// TIA Portal V16 program export: 3 tag tables, 0 data types, 6 data blocks, 22 code blocks (in call order from the OBs), 35 instance data blocks

VAR_GLOBAL   // PLC tag table "Default tag table"
   EDGE_1 AT %M100.0 : Bool;
   EDGE_2 AT %M100.1 : Bool;
   System_Byte AT %MB1 : Byte;
   FirstScan AT %M1.0 : Bool;
   DiagStatusUpdate AT %M1.1 : Bool;
   AlwaysTRUE AT %M1.2 : Bool;
   AlwaysFALSE AT %M1.3 : Bool;
   Clock_Byte AT %MB0 : Byte;
   Clock_10Hz AT %M0.0 : Bool;
   Clock_5Hz AT %M0.1 : Bool;
   "Clock_2.5Hz" AT %M0.2 : Bool;
   Clock_2Hz AT %M0.3 : Bool;
   "Clock_1.25Hz" AT %M0.4 : Bool;
   Clock_1Hz AT %M0.5 : Bool;
   "Clock_0.625Hz" AT %M0.6 : Bool;
   "Clock_0.5Hz" AT %M0.7 : Bool;
   EDGE_3 AT %M100.2 : Bool;
   EDGE_4 AT %M100.3 : Bool;
   RET_VAL_SYSTEM_TIME AT %MW102 : Word;
   EDGE_5 AT %M100.4 : Bool;
   EDGE_6 AT %M100.5 : Bool;
   EDGE_7 AT %M100.6 : Bool;
END_VAR

VAR_GLOBAL   // PLC tag table "Inputs"
   "EV1.1_ABERTA" AT %I0.0 : Bool;
   "EV1.1_FECHADA" AT %I0.1 : Bool;
   "EV2.1_ABERTA" AT %I0.2 : Bool;
   "EV2.1_FECHADA" AT %I0.3 : Bool;
   "EV3.1_ABERTA" AT %I0.4 : Bool;
   "EV3.1_FECHADA" AT %I0.5 : Bool;
   "EV4.1_ABERTA" AT %I0.6 : Bool;
   "EV4.1_FECHADA" AT %I0.7 : Bool;
   "EV5.1_ABERTA" AT %I1.0 : Bool;
   "EV5.1_FECHADA" AT %I1.1 : Bool;
   "EV1.2_ABERTA" AT %I1.2 : Bool;
   "EV1.2_FECHADA" AT %I1.3 : Bool;
   "EV2.2_ABERTA" AT %I1.4 : Bool;
   "EV2.2_FECHADA" AT %I1.5 : Bool;
   "EV3.2_ABERTA" AT %I2.0 : Bool;
   "EV3.2_FECHADA" AT %I2.1 : Bool;
   "EV4.2_ABERTA" AT %I2.2 : Bool;
   "EV4.2_FECHADA" AT %I2.3 : Bool;
   "EV5.2_ABERTA" AT %I2.4 : Bool;
   "EV5.2_FECHADA" AT %I2.5 : Bool;
   PRESSOSTATO_1 AT %IW4 : Word;
   PRESSOSTATO_2 AT %IW6 : Word;
   AVARIA_BOMBA_1 AT %I2.6 : Bool;
   AVARIA_BOMBA_2 AT %I2.7 : Bool;
   AVARIA_BOMBA_3 AT %I3.0 : Bool;
END_VAR

VAR_GLOBAL   // PLC tag table "Outputs"
   "EV1.1" AT %Q0.0 : Bool;
   "EV2.1" AT %Q0.1 : Bool;
   "EV3.1" AT %Q0.2 : Bool;
   "EV4.1" AT %Q0.3 : Bool;
   "EV5.1" AT %Q0.4 : Bool;
   "EV1.2" AT %Q0.5 : Bool;
   "EV2.2" AT %Q0.6 : Bool;
   "EV3.2" AT %Q0.7 : Bool;
   "EV4.2" AT %Q1.0 : Bool;
   "EV5.2" AT %Q1.1 : Bool;
   BOMBA_1_VAR AT %Q2.0 : Bool;
   BOMBA_2_VAR AT %Q2.1 : Bool;
   BOMBA_3_RESERVA AT %Q2.2 : Bool;
   ULTRAVIOLETA AT %Q2.3 : Bool;
END_VAR

DATA_BLOCK "Dados_Bombas"   // DB11
{ S7_Optimized_Access := 'TRUE' }
VERSION : 0.1
// stored: AutoNumber true, IsOnlyStoredInLoadMemory false, IsRetainMemResEnabled false, IsWriteProtectedInAS false, MemoryReserve 100
   VAR
      CONV_T_ALTERNANCIA_BOMBAS : Time;
      HORAS_TON_B2 : Int;
      HORAS_TON_B3 : Int;
      HORAS_TON_B1 : Int;
   END_VAR
BEGIN
END_DATA_BLOCK

DATA_BLOCK "Estados_HMI"   // DB18
{ S7_Optimized_Access := 'TRUE' }
VERSION : 0.1
// stored: AutoNumber true, IsOnlyStoredInLoadMemory false, IsRetainMemResEnabled false, IsWriteProtectedInAS false, MemoryReserve 100
   VAR
      "EV1.1_ESTADO" : Int;
      "EV2.1_ESTADO" : Int;
      "EV3.1_ESTADO" : Int;
      "EV4.1_ESTADO" : Int;
      "EV5.1_ESTADO" : Int;
      "EV1.2_ESTADO" : Int;
      "EV2.2_ESTADO" : Int;
      "EV3.2_ESTADO" : Int;
      "EV4.2_ESTADO" : Int;
      "EV5.2_ESTADO" : Int;
      "EV1.1_ESTADO_PAGCMD" : Int;
      "EV2.1_ESTADO_PAGCMD" : Int;
      "EV3.1_ESTADO_PAGCMD" : Int;
      "EV4.1_ESTADO_PAGCMD" : Int;
      "EV5.1_ESTADO_PAGCMD" : Int;
      "EV1.2_ESTADO_PAGCMD" : Int;
      "EV2.2_ESTADO_PAGCMD" : Int;
      "EV3.2_ESTADO_PAGCMD" : Int;
      "EV4.2_ESTADO_PAGCMD" : Int;
      "EV5.2_ESTADO_PAGCMD" : Int;
      BOMBA_1_ESTADO : Int;
      BOMBA_2_ESTADO : Int;
      BOMBA_3_ESTADO : Int;
      BOMBA_1_ESTADO_PAGCMD : Int;
      BOMBA_2_ESTADO_PAGCMD : Int;
      BOMBA_3_ESTADO_PAGCMD : Int;
      T_LAV_MINUTOS : Int;
      T_RINSE_MINUTOS : Int;
      ALARMES_LISTA_1 : Word;
      ALARMES_LISTA_2 : Word;
      ALARMES_LISTA_3 : Word;
   END_VAR
BEGIN
END_DATA_BLOCK

DATA_BLOCK "Inputs_HMI"   // DB6
{ S7_Optimized_Access := 'TRUE' }
VERSION : 0.1
// stored: AutoNumber true, IsOnlyStoredInLoadMemory false, IsRetainMemResEnabled false, IsWriteProtectedInAS false, MemoryReserve 100
   VAR RETAIN
      T_LAVAGEM : Time;
      T_RINSE : Time;
      T_STOP_BOMBAS : Time;
      T_POS_EVS : Time;
      ENABLE_CICLO_FILT1 : Bool;
      ENABLE_CICLO_FILT2 : Bool;
   END_VAR
   VAR
      START_CICLO_FILT1 : Bool;
      START_CICLO_FILT2 : Bool;
      STOP_CICLO : Bool;
      REARME : Bool;
      "MAN/AUTO" : Bool;
      "ON_OFF_EV1.1" : Bool;
      "ON_OFF_EV2.1" : Bool;
      "ON_OFF_EV3.1" : Bool;
      "ON_OFF_EV4.1" : Bool;
      "ON_OFF_EV5.1" : Bool;
      "ON_OFF_EV1.2" : Bool;
      "ON_OFF_EV2.2" : Bool;
      "ON_OFF_EV3.2" : Bool;
      "ON_OFF_EV4.2" : Bool;
      "ON_OFF_EV5.2" : Bool;
   END_VAR
   VAR RETAIN
      "MAN/AUTO_BOMBAS" : Bool;
      T_ALTERNANCIA_BOMBAS : Real;
   END_VAR
   VAR
      ON_OFF_BOMBA_1 : Bool;
      ON_OFF_BOMBA_2 : Bool;
      ON_OFF_BOMBA_3 : Bool;
      RESET_CNT_B1 : Bool;
      RESET_CNT_B2 : Bool;
      RESET_CNT_B3 : Bool;
   END_VAR
   VAR RETAIN
      SP_PRESS_FILT1 : Real;
      SP_PRESS_FILT2 : Real;
   END_VAR
BEGIN
END_DATA_BLOCK

DATA_BLOCK "Dados_Ciclo"   // DB7
{ S7_Optimized_Access := 'TRUE' }
VERSION : 0.1
// stored: AutoNumber true, IsOnlyStoredInLoadMemory false, IsRetainMemResEnabled false, IsWriteProtectedInAS false, MemoryReserve 100
   VAR
      HOLD_ETAPA_1 : Bool;
   END_VAR
   VAR RETAIN
      FILTRO1_EM_CICLO : Bool;
      FILTRO2_EM_CICLO : Bool;
      FECHO_FILT_1 : Bool;
      FECHO_FILT_2 : Bool;
      ETAPA_ANTERIOR : Int := 1;
   END_VAR
   VAR
      ETAPA_N : Bool;
      POS_EVS_FILT_1 : String;
      POS_EVS_FILT_2 : String;
      PRESS_SP_FILT_1 : Bool;
      PRESS_SP_FILT_2 : Bool;
   END_VAR
   VAR RETAIN
      STOP_CICLO : Bool;
   END_VAR
   VAR
      AGEND_FILT_1 : Bool;
      AGEND_FILT_2 : Bool;
   END_VAR
   VAR RETAIN
      HORA_INIC_FILT_1 : USInt;
      MIN_INIC_FILT_1 : USInt;
      HORA_INIC_FILT_2 : USInt;
      MIN_INIC_FILT_2 : USInt;
      ENABLE_AGEND_FILT_1 : Bool;
      ENABLE_AGEND_FILT_2 : Bool;
   END_VAR
   VAR
      PRESSÃO_FILT1 : Real;
      PRESSÃO_FILT2 : Real;
   END_VAR
BEGIN
END_DATA_BLOCK

DATA_BLOCK "Etapas_Grafcet"   // DB1
{ S7_Optimized_Access := 'TRUE' }
VERSION : 0.1
// stored: AutoNumber true, IsOnlyStoredInLoadMemory false, IsRetainMemResEnabled false, IsWriteProtectedInAS false, MemoryReserve 100
   VAR
      ETAPA_1 : Bool;
      ETAPA_2 : Bool;
      ETAPA_3 : Bool;
      ETAPA_4 : Bool;
      ETAPA_5 : Bool;
      ETAPA_6 : Bool;
      ETAPA_7 : Bool;
      ETAPA_8 : Bool;
      ETAPA_9 : Bool;
      ETAPA_10 : Bool;
      ETAPA_11 : Bool;
      ETAPA_12 : Bool;
      ETAPA_13 : Bool;
      ETAPA_14 : Bool;
      ETAPA_15 : Bool := true;
      ETAPA_16 : Bool;
   END_VAR
BEGIN
END_DATA_BLOCK

DATA_BLOCK "System_Time"   // DB40
{ S7_Optimized_Access := 'TRUE' }
VERSION : 0.1
// stored: AutoNumber true, IsOnlyStoredInLoadMemory false, IsRetainMemResEnabled false, IsWriteProtectedInAS false, MemoryReserve 100
   VAR
      REAL_TIME_DATA : DTL;
   END_VAR
BEGIN
END_DATA_BLOCK

ORGANIZATION_BLOCK "Main"   // OB1, LAD, ProgramCycle
TITLE = "Main Program Sweep (Cycle)"
{ S7_Optimized_Access := 'TRUE' }
VERSION : 0.1
// stored: AutoNumber true, IsIECCheckEnabled false, SetENOAutomatically false
   VAR_INPUT
      Initial_Call : Bool;   // Initial call of this OB
      Remanence : Bool;   // =True, if remanent data are available
   END_VAR
   VAR_TEMP   // added for the SCL form of the ladder/FBD networks
      _w1 : Bool;
   END_VAR
BEGIN

REGION Network 1: Ciclo de lavagem e enxaguamento
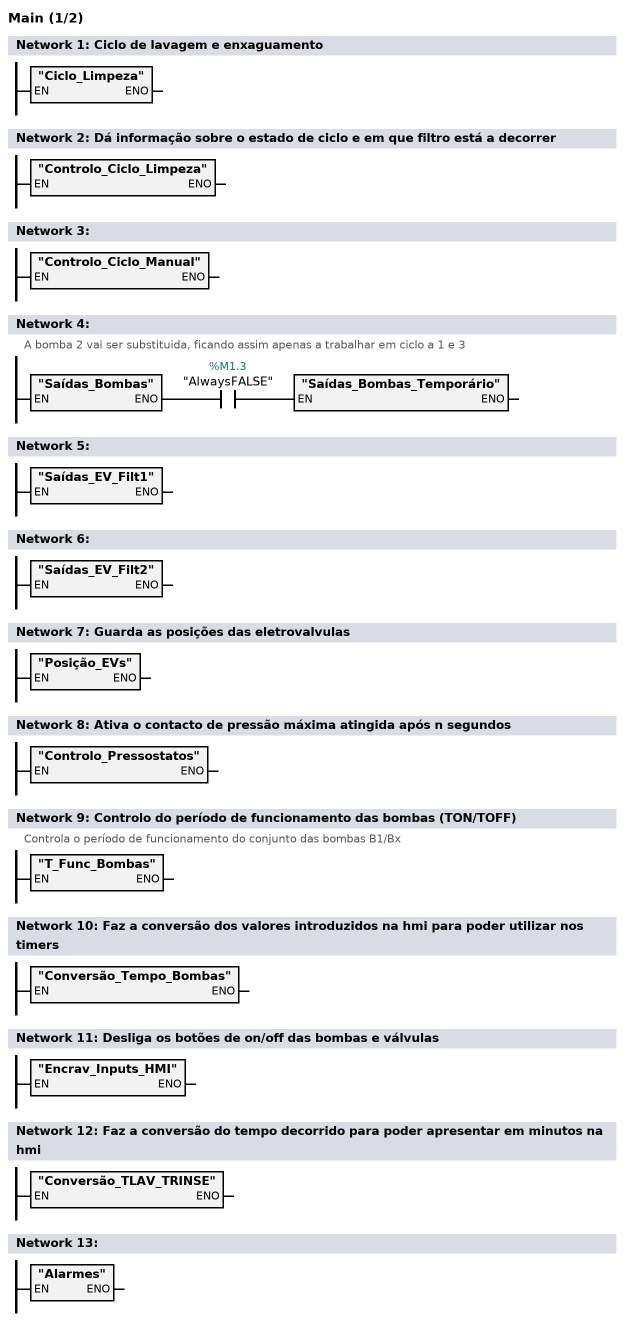
   RUNG wire#powerrail
      "Ciclo_Limpeza"()
   END_RUNG
   // the same network as SCL:
   "Ciclo_Limpeza"();
END_REGION

REGION Network 2: Dá informação sobre o estado de ciclo e em que filtro está a decorrer
   RUNG wire#powerrail
      "Controlo_Ciclo_Limpeza"()
   END_RUNG
   // the same network as SCL:
   "Controlo_Ciclo_Limpeza"();
END_REGION

REGION Network 3
   RUNG wire#powerrail
      "Controlo_Ciclo_Manual"()
   END_RUNG
   // the same network as SCL:
   "Controlo_Ciclo_Manual"();
END_REGION

REGION Network 4
   // A bomba 2 vai ser substituida, ficando assim apenas a trabalhar em ciclo a 1 e 3
   RUNG wire#powerrail
      "Saídas_Bombas"()
      Contact( "AlwaysFALSE" )
      "Saídas_Bombas_Temporário"()
   END_RUNG
   // the same network as SCL:
   "Saídas_Bombas"(ENO => #_w1);
   IF #_w1 AND "AlwaysFALSE" THEN "Saídas_Bombas_Temporário"(); END_IF;
END_REGION

REGION Network 5
   RUNG wire#powerrail
      "Saídas_EV_Filt1"()
   END_RUNG
   // the same network as SCL:
   "Saídas_EV_Filt1"();
END_REGION

REGION Network 6
   RUNG wire#powerrail
      "Saídas_EV_Filt2"()
   END_RUNG
   // the same network as SCL:
   "Saídas_EV_Filt2"();
END_REGION

REGION Network 7: Guarda as posições das eletrovalvulas
   RUNG wire#powerrail
      "Posição_EVs"()
   END_RUNG
   // the same network as SCL:
   "Posição_EVs"();
END_REGION

REGION Network 8: Ativa o contacto de pressão máxima atingida após n segundos
   RUNG wire#powerrail
      "Controlo_Pressostatos"()
   END_RUNG
   // the same network as SCL:
   "Controlo_Pressostatos"();
END_REGION

REGION Network 9: Controlo do período de funcionamento das bombas (TON/TOFF)
   // Controla o período de funcionamento do conjunto das bombas B1/Bx
   RUNG wire#powerrail
      "T_Func_Bombas"()
   END_RUNG
   // the same network as SCL:
   "T_Func_Bombas"();
END_REGION

REGION Network 10: Faz a conversão dos valores introduzidos na hmi para poder utilizar nos timers
   RUNG wire#powerrail
      "Conversão_Tempo_Bombas"()
   END_RUNG
   // the same network as SCL:
   "Conversão_Tempo_Bombas"();
END_REGION

REGION Network 11: Desliga os botões de on/off das bombas e válvulas
   RUNG wire#powerrail
      "Encrav_Inputs_HMI"()
   END_RUNG
   // the same network as SCL:
   "Encrav_Inputs_HMI"();
END_REGION

REGION Network 12: Faz a conversão do tempo decorrido para poder apresentar em minutos na hmi
   RUNG wire#powerrail
      "Conversão_TLAV_TRINSE"()
   END_RUNG
   // the same network as SCL:
   "Conversão_TLAV_TRINSE"();
END_REGION

REGION Network 13
   RUNG wire#powerrail
      "Alarmes"()
   END_RUNG
   // the same network as SCL:
   "Alarmes"();
END_REGION

REGION Network 14: Ultravioleta
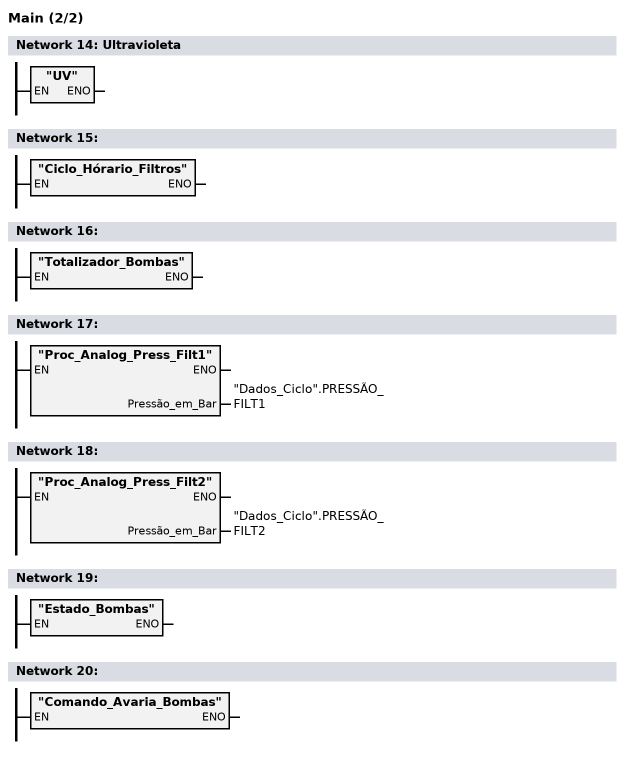
   RUNG wire#powerrail
      "UV"()
   END_RUNG
   // the same network as SCL:
   "UV"();
END_REGION

REGION Network 15
   RUNG wire#powerrail
      "Ciclo_Hórario_Filtros"()
   END_RUNG
   // the same network as SCL:
   "Ciclo_Hórario_Filtros"();
END_REGION

REGION Network 16
   RUNG wire#powerrail
      "Totalizador_Bombas"()
   END_RUNG
   // the same network as SCL:
   "Totalizador_Bombas"();
END_REGION

REGION Network 17
   RUNG wire#powerrail
      "Proc_Analog_Press_Filt1"(Pressão_em_Bar => "Dados_Ciclo".PRESSÃO_FILT1)
   END_RUNG
   // the same network as SCL:
   "Proc_Analog_Press_Filt1"(Pressão_em_Bar => "Dados_Ciclo".PRESSÃO_FILT1);
END_REGION

REGION Network 18
   RUNG wire#powerrail
      "Proc_Analog_Press_Filt2"(Pressão_em_Bar => "Dados_Ciclo".PRESSÃO_FILT2)
   END_RUNG
   // the same network as SCL:
   "Proc_Analog_Press_Filt2"(Pressão_em_Bar => "Dados_Ciclo".PRESSÃO_FILT2);
END_REGION

REGION Network 19
   RUNG wire#powerrail
      "Estado_Bombas"()
   END_RUNG
   // the same network as SCL:
   "Estado_Bombas"();
END_REGION

REGION Network 20
   RUNG wire#powerrail
      "Comando_Avaria_Bombas"()
   END_RUNG
   // the same network as SCL:
   "Comando_Avaria_Bombas"();
END_REGION
END_ORGANIZATION_BLOCK

FUNCTION "Ciclo_Limpeza" : Void   // FC1, LAD
TITLE = Ciclo de lavagem e enxaguamento
{ S7_Optimized_Access := 'TRUE' }
VERSION : 0.1
// stored: AutoNumber true, IsIECCheckEnabled false, SetENOAutomatically false, UDAEnableTagReadback false
   VAR_TEMP   // added for the SCL form of the ladder/FBD networks
      _w1 : Bool;
      _w2 : Bool;
      _w3 : Bool;
   END_VAR
BEGIN

REGION Network 1: Etapa 1 (Início)
   // Início com EV's na posição de filtração. As bombas podem estar ligadas ou não, conforme a posição do switch 4
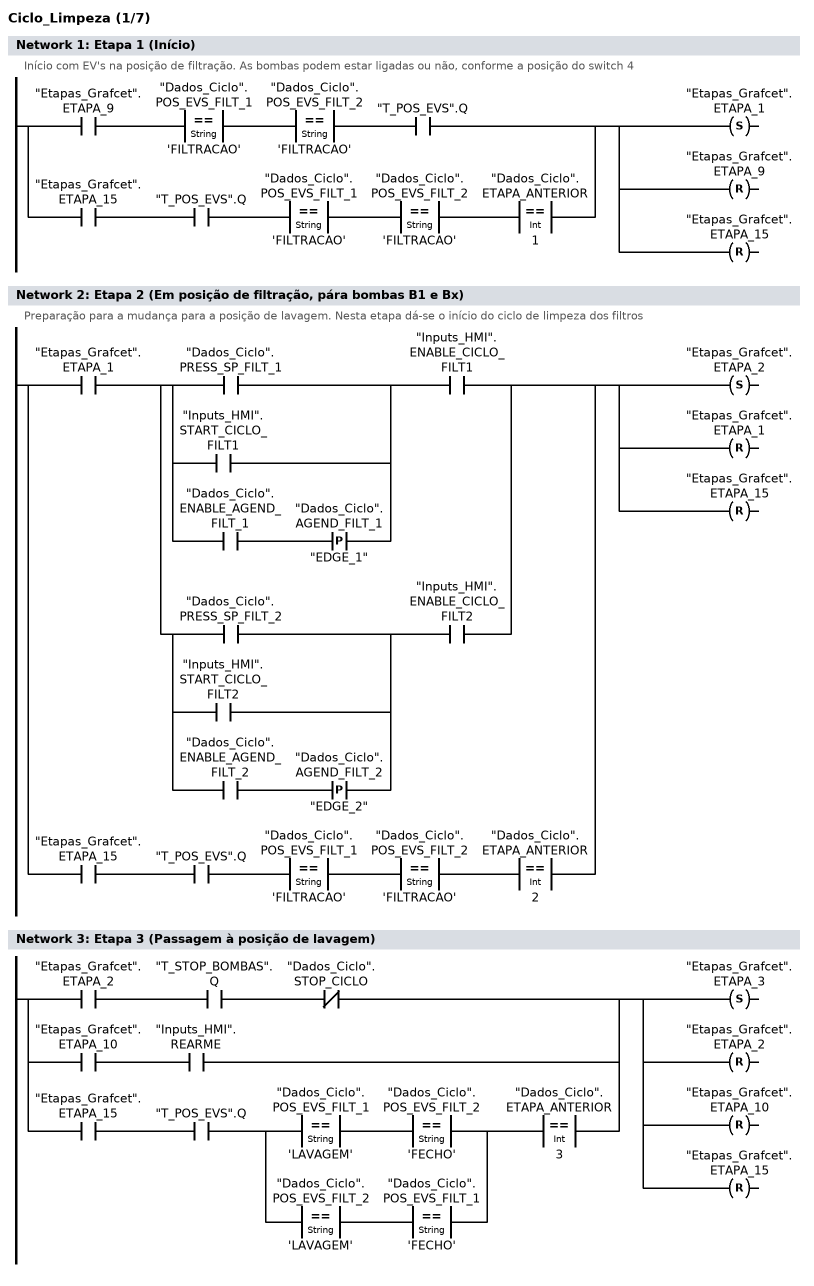
   RUNG wire#powerrail
      Contact( "Etapas_Grafcet".ETAPA_9 )
      { S7_Templates := "SrcType := String" } EQ_Contact(in1 := "Dados_Ciclo".POS_EVS_FILT_1, in2 := 'FILTRACAO')
      { S7_Templates := "SrcType := String" } EQ_Contact(in1 := "Dados_Ciclo".POS_EVS_FILT_2, in2 := 'FILTRACAO')
      Contact( "T_POS_EVS".Q )
      wire#w1
      S_Coil( "Etapas_Grafcet".ETAPA_1 )
   END_RUNG
   RUNG wire#powerrail
      Contact( "Etapas_Grafcet".ETAPA_15 )
      Contact( "T_POS_EVS".Q )
      { S7_Templates := "SrcType := String" } EQ_Contact(in1 := "Dados_Ciclo".POS_EVS_FILT_1, in2 := 'FILTRACAO')
      { S7_Templates := "SrcType := String" } EQ_Contact(in1 := "Dados_Ciclo".POS_EVS_FILT_2, in2 := 'FILTRACAO')
      { S7_Templates := "SrcType := Int" } EQ_Contact(in1 := "Dados_Ciclo".ETAPA_ANTERIOR, in2 := 1)
   END_RUNG wire#w1
   RUNG wire#w1
      R_Coil( "Etapas_Grafcet".ETAPA_9 )
   END_RUNG
   RUNG wire#w1
      R_Coil( "Etapas_Grafcet".ETAPA_15 )
   END_RUNG
   // the same network as SCL:
   IF ("Etapas_Grafcet".ETAPA_9 AND ("Dados_Ciclo".POS_EVS_FILT_1 = 'FILTRACAO') AND ("Dados_Ciclo".POS_EVS_FILT_2 = 'FILTRACAO') AND "T_POS_EVS".Q) OR ("Etapas_Grafcet".ETAPA_15 AND "T_POS_EVS".Q AND ("Dados_Ciclo".POS_EVS_FILT_1 = 'FILTRACAO') AND ("Dados_Ciclo".POS_EVS_FILT_2 = 'FILTRACAO') AND ("Dados_Ciclo".ETAPA_ANTERIOR = 1)) THEN
       "Etapas_Grafcet".ETAPA_1 := TRUE;
   END_IF;
   #_w1 := ("Etapas_Grafcet".ETAPA_9 AND ("Dados_Ciclo".POS_EVS_FILT_1 = 'FILTRACAO') AND ("Dados_Ciclo".POS_EVS_FILT_2 = 'FILTRACAO') AND "T_POS_EVS".Q) OR ("Etapas_Grafcet".ETAPA_15 AND "T_POS_EVS".Q AND ("Dados_Ciclo".POS_EVS_FILT_1 = 'FILTRACAO') AND ("Dados_Ciclo".POS_EVS_FILT_2 = 'FILTRACAO') AND ("Dados_Ciclo".ETAPA_ANTERIOR = 1));
   IF #_w1 THEN
       "Etapas_Grafcet".ETAPA_9 := FALSE;
       "Etapas_Grafcet".ETAPA_15 := FALSE;
   END_IF;
END_REGION

REGION Network 2: Etapa 2 (Em posição de filtração, pára bombas B1 e Bx)
   // Preparação para a mudança para a posição de lavagem. Nesta etapa dá-se o início do ciclo de limpeza dos filtros
   RUNG wire#powerrail
      Contact( "Etapas_Grafcet".ETAPA_1 )
      wire#w1
      Contact( "Dados_Ciclo".PRESS_SP_FILT_1 )
      wire#w2
      Contact( "Inputs_HMI".ENABLE_CICLO_FILT1 )
      wire#w3
      S_Coil( "Etapas_Grafcet".ETAPA_2 )
   END_RUNG
   RUNG wire#w1
      Contact( "Inputs_HMI".START_CICLO_FILT1 )
   END_RUNG wire#w2
   RUNG wire#w1
      Contact( "Dados_Ciclo".ENABLE_AGEND_FILT_1 )
      P_Contact(operand := "Dados_Ciclo".AGEND_FILT_1, bit := "EDGE_1")
   END_RUNG wire#w2
   RUNG wire#w1
      Contact( "Dados_Ciclo".PRESS_SP_FILT_2 )
      wire#w4
      Contact( "Inputs_HMI".ENABLE_CICLO_FILT2 )
   END_RUNG wire#w3
   RUNG wire#w1
      Contact( "Inputs_HMI".START_CICLO_FILT2 )
   END_RUNG wire#w4
   RUNG wire#w1
      Contact( "Dados_Ciclo".ENABLE_AGEND_FILT_2 )
      P_Contact(operand := "Dados_Ciclo".AGEND_FILT_2, bit := "EDGE_2")
   END_RUNG wire#w4
   RUNG wire#powerrail
      Contact( "Etapas_Grafcet".ETAPA_15 )
      Contact( "T_POS_EVS".Q )
      { S7_Templates := "SrcType := String" } EQ_Contact(in1 := "Dados_Ciclo".POS_EVS_FILT_1, in2 := 'FILTRACAO')
      { S7_Templates := "SrcType := String" } EQ_Contact(in1 := "Dados_Ciclo".POS_EVS_FILT_2, in2 := 'FILTRACAO')
      { S7_Templates := "SrcType := Int" } EQ_Contact(in1 := "Dados_Ciclo".ETAPA_ANTERIOR, in2 := 2)
   END_RUNG wire#w3
   RUNG wire#w3
      R_Coil( "Etapas_Grafcet".ETAPA_1 )
   END_RUNG
   RUNG wire#w3
      R_Coil( "Etapas_Grafcet".ETAPA_15 )
   END_RUNG
   // the same network as SCL:
   #_w1 := "Etapas_Grafcet".ETAPA_1 AND "Dados_Ciclo".ENABLE_AGEND_FILT_1 AND "Dados_Ciclo".AGEND_FILT_1 AND NOT "EDGE_1";   // rising edge of "Dados_Ciclo".AGEND_FILT_1
   "EDGE_1" := "Dados_Ciclo".AGEND_FILT_1;
   #_w2 := "Etapas_Grafcet".ETAPA_1 AND "Dados_Ciclo".ENABLE_AGEND_FILT_2 AND "Dados_Ciclo".AGEND_FILT_2 AND NOT "EDGE_2";   // rising edge of "Dados_Ciclo".AGEND_FILT_2
   "EDGE_2" := "Dados_Ciclo".AGEND_FILT_2;
   IF ((("Etapas_Grafcet".ETAPA_1 AND ("Dados_Ciclo".PRESS_SP_FILT_1 OR "Inputs_HMI".START_CICLO_FILT1)) OR #_w1) AND "Inputs_HMI".ENABLE_CICLO_FILT1) OR ((("Etapas_Grafcet".ETAPA_1 AND ("Dados_Ciclo".PRESS_SP_FILT_2 OR "Inputs_HMI".START_CICLO_FILT2)) OR #_w2) AND "Inputs_HMI".ENABLE_CICLO_FILT2) OR ("Etapas_Grafcet".ETAPA_15 AND "T_POS_EVS".Q AND ("Dados_Ciclo".POS_EVS_FILT_1 = 'FILTRACAO') AND ("Dados_Ciclo".POS_EVS_FILT_2 = 'FILTRACAO') AND ("Dados_Ciclo".ETAPA_ANTERIOR = 2)) THEN
       "Etapas_Grafcet".ETAPA_2 := TRUE;
   END_IF;
   #_w3 := ((("Etapas_Grafcet".ETAPA_1 AND ("Dados_Ciclo".PRESS_SP_FILT_1 OR "Inputs_HMI".START_CICLO_FILT1)) OR #_w1) AND "Inputs_HMI".ENABLE_CICLO_FILT1) OR ((("Etapas_Grafcet".ETAPA_1 AND ("Dados_Ciclo".PRESS_SP_FILT_2 OR "Inputs_HMI".START_CICLO_FILT2)) OR #_w2) AND "Inputs_HMI".ENABLE_CICLO_FILT2) OR ("Etapas_Grafcet".ETAPA_15 AND "T_POS_EVS".Q AND ("Dados_Ciclo".POS_EVS_FILT_1 = 'FILTRACAO') AND ("Dados_Ciclo".POS_EVS_FILT_2 = 'FILTRACAO') AND ("Dados_Ciclo".ETAPA_ANTERIOR = 2));
   IF #_w3 THEN
       "Etapas_Grafcet".ETAPA_1 := FALSE;
       "Etapas_Grafcet".ETAPA_15 := FALSE;
   END_IF;
END_REGION

REGION Network 3: Etapa 3 (Passagem à posição de lavagem)
   RUNG wire#powerrail
      Contact( "Etapas_Grafcet".ETAPA_2 )
      Contact( "T_STOP_BOMBAS".Q )
      I_Contact( "Dados_Ciclo".STOP_CICLO )
      wire#w1
      S_Coil( "Etapas_Grafcet".ETAPA_3 )
   END_RUNG
   RUNG wire#powerrail
      Contact( "Etapas_Grafcet".ETAPA_10 )
      Contact( "Inputs_HMI".REARME )
   END_RUNG wire#w1
   RUNG wire#powerrail
      Contact( "Etapas_Grafcet".ETAPA_15 )
      Contact( "T_POS_EVS".Q )
      wire#w2
      { S7_Templates := "SrcType := String" } EQ_Contact(in1 := "Dados_Ciclo".POS_EVS_FILT_1, in2 := 'LAVAGEM')
      { S7_Templates := "SrcType := String" } EQ_Contact(in1 := "Dados_Ciclo".POS_EVS_FILT_2, in2 := 'FECHO')
      wire#w3
      { S7_Templates := "SrcType := Int" } EQ_Contact(in1 := "Dados_Ciclo".ETAPA_ANTERIOR, in2 := 3)
   END_RUNG wire#w1
   RUNG wire#w2
      { S7_Templates := "SrcType := String" } EQ_Contact(in1 := "Dados_Ciclo".POS_EVS_FILT_2, in2 := 'LAVAGEM')
      { S7_Templates := "SrcType := String" } EQ_Contact(in1 := "Dados_Ciclo".POS_EVS_FILT_1, in2 := 'FECHO')
   END_RUNG wire#w3
   RUNG wire#w1
      R_Coil( "Etapas_Grafcet".ETAPA_2 )
   END_RUNG
   RUNG wire#w1
      R_Coil( "Etapas_Grafcet".ETAPA_10 )
   END_RUNG
   RUNG wire#w1
      R_Coil( "Etapas_Grafcet".ETAPA_15 )
   END_RUNG
   // the same network as SCL:
   IF ("Etapas_Grafcet".ETAPA_2 AND "T_STOP_BOMBAS".Q AND NOT "Dados_Ciclo".STOP_CICLO) OR ("Etapas_Grafcet".ETAPA_10 AND "Inputs_HMI".REARME) OR ("Etapas_Grafcet".ETAPA_15 AND "T_POS_EVS".Q AND ((("Dados_Ciclo".POS_EVS_FILT_1 = 'LAVAGEM') AND ("Dados_Ciclo".POS_EVS_FILT_2 = 'FECHO')) OR (("Dados_Ciclo".POS_EVS_FILT_2 = 'LAVAGEM') AND ("Dados_Ciclo".POS_EVS_FILT_1 = 'FECHO'))) AND ("Dados_Ciclo".ETAPA_ANTERIOR = 3)) THEN
       "Etapas_Grafcet".ETAPA_3 := TRUE;
   END_IF;
   #_w1 := ("Etapas_Grafcet".ETAPA_2 AND "T_STOP_BOMBAS".Q AND NOT "Dados_Ciclo".STOP_CICLO) OR ("Etapas_Grafcet".ETAPA_10 AND "Inputs_HMI".REARME) OR ("Etapas_Grafcet".ETAPA_15 AND "T_POS_EVS".Q AND ((("Dados_Ciclo".POS_EVS_FILT_1 = 'LAVAGEM') AND ("Dados_Ciclo".POS_EVS_FILT_2 = 'FECHO')) OR (("Dados_Ciclo".POS_EVS_FILT_2 = 'LAVAGEM') AND ("Dados_Ciclo".POS_EVS_FILT_1 = 'FECHO'))) AND ("Dados_Ciclo".ETAPA_ANTERIOR = 3));
   IF #_w1 THEN
       "Etapas_Grafcet".ETAPA_2 := FALSE;
       "Etapas_Grafcet".ETAPA_10 := FALSE;
       "Etapas_Grafcet".ETAPA_15 := FALSE;
   END_IF;
END_REGION

REGION Network 4: Etapa 4 (Em lavagem, B1 e BX ligadas)
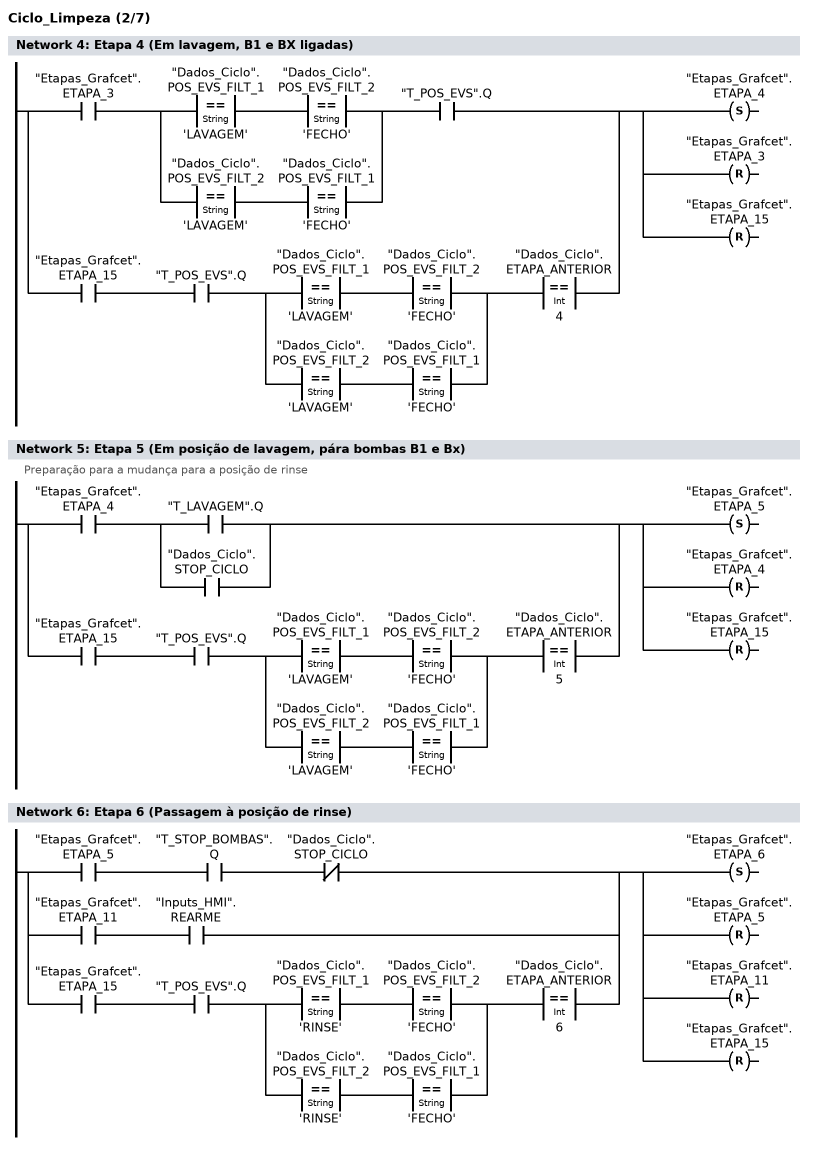
   RUNG wire#powerrail
      Contact( "Etapas_Grafcet".ETAPA_3 )
      wire#w1
      { S7_Templates := "SrcType := String" } EQ_Contact(in1 := "Dados_Ciclo".POS_EVS_FILT_1, in2 := 'LAVAGEM')
      { S7_Templates := "SrcType := String" } EQ_Contact(in1 := "Dados_Ciclo".POS_EVS_FILT_2, in2 := 'FECHO')
      wire#w2
      Contact( "T_POS_EVS".Q )
      wire#w3
      S_Coil( "Etapas_Grafcet".ETAPA_4 )
   END_RUNG
   RUNG wire#w1
      { S7_Templates := "SrcType := String" } EQ_Contact(in1 := "Dados_Ciclo".POS_EVS_FILT_2, in2 := 'LAVAGEM')
      { S7_Templates := "SrcType := String" } EQ_Contact(in1 := "Dados_Ciclo".POS_EVS_FILT_1, in2 := 'FECHO')
   END_RUNG wire#w2
   RUNG wire#powerrail
      Contact( "Etapas_Grafcet".ETAPA_15 )
      Contact( "T_POS_EVS".Q )
      wire#w4
      { S7_Templates := "SrcType := String" } EQ_Contact(in1 := "Dados_Ciclo".POS_EVS_FILT_1, in2 := 'LAVAGEM')
      { S7_Templates := "SrcType := String" } EQ_Contact(in1 := "Dados_Ciclo".POS_EVS_FILT_2, in2 := 'FECHO')
      wire#w5
      { S7_Templates := "SrcType := Int" } EQ_Contact(in1 := "Dados_Ciclo".ETAPA_ANTERIOR, in2 := 4)
   END_RUNG wire#w3
   RUNG wire#w4
      { S7_Templates := "SrcType := String" } EQ_Contact(in1 := "Dados_Ciclo".POS_EVS_FILT_2, in2 := 'LAVAGEM')
      { S7_Templates := "SrcType := String" } EQ_Contact(in1 := "Dados_Ciclo".POS_EVS_FILT_1, in2 := 'FECHO')
   END_RUNG wire#w5
   RUNG wire#w3
      R_Coil( "Etapas_Grafcet".ETAPA_3 )
   END_RUNG
   RUNG wire#w3
      R_Coil( "Etapas_Grafcet".ETAPA_15 )
   END_RUNG
   // the same network as SCL:
   IF ("Etapas_Grafcet".ETAPA_3 AND ((("Dados_Ciclo".POS_EVS_FILT_1 = 'LAVAGEM') AND ("Dados_Ciclo".POS_EVS_FILT_2 = 'FECHO')) OR (("Dados_Ciclo".POS_EVS_FILT_2 = 'LAVAGEM') AND ("Dados_Ciclo".POS_EVS_FILT_1 = 'FECHO'))) AND "T_POS_EVS".Q) OR ("Etapas_Grafcet".ETAPA_15 AND "T_POS_EVS".Q AND ((("Dados_Ciclo".POS_EVS_FILT_1 = 'LAVAGEM') AND ("Dados_Ciclo".POS_EVS_FILT_2 = 'FECHO')) OR (("Dados_Ciclo".POS_EVS_FILT_2 = 'LAVAGEM') AND ("Dados_Ciclo".POS_EVS_FILT_1 = 'FECHO'))) AND ("Dados_Ciclo".ETAPA_ANTERIOR = 4)) THEN
       "Etapas_Grafcet".ETAPA_4 := TRUE;
   END_IF;
   #_w1 := ("Etapas_Grafcet".ETAPA_3 AND ((("Dados_Ciclo".POS_EVS_FILT_1 = 'LAVAGEM') AND ("Dados_Ciclo".POS_EVS_FILT_2 = 'FECHO')) OR (("Dados_Ciclo".POS_EVS_FILT_2 = 'LAVAGEM') AND ("Dados_Ciclo".POS_EVS_FILT_1 = 'FECHO'))) AND "T_POS_EVS".Q) OR ("Etapas_Grafcet".ETAPA_15 AND "T_POS_EVS".Q AND ((("Dados_Ciclo".POS_EVS_FILT_1 = 'LAVAGEM') AND ("Dados_Ciclo".POS_EVS_FILT_2 = 'FECHO')) OR (("Dados_Ciclo".POS_EVS_FILT_2 = 'LAVAGEM') AND ("Dados_Ciclo".POS_EVS_FILT_1 = 'FECHO'))) AND ("Dados_Ciclo".ETAPA_ANTERIOR = 4));
   IF #_w1 THEN
       "Etapas_Grafcet".ETAPA_3 := FALSE;
       "Etapas_Grafcet".ETAPA_15 := FALSE;
   END_IF;
END_REGION

REGION Network 5: Etapa 5 (Em posição de lavagem, pára bombas B1 e Bx)
   // Preparação para a mudança para a posição de rinse
   RUNG wire#powerrail
      Contact( "Etapas_Grafcet".ETAPA_4 )
      wire#w1
      Contact( "T_LAVAGEM".Q )
      wire#w2
      S_Coil( "Etapas_Grafcet".ETAPA_5 )
   END_RUNG
   RUNG wire#w1
      Contact( "Dados_Ciclo".STOP_CICLO )
   END_RUNG wire#w2
   RUNG wire#powerrail
      Contact( "Etapas_Grafcet".ETAPA_15 )
      Contact( "T_POS_EVS".Q )
      wire#w3
      { S7_Templates := "SrcType := String" } EQ_Contact(in1 := "Dados_Ciclo".POS_EVS_FILT_1, in2 := 'LAVAGEM')
      { S7_Templates := "SrcType := String" } EQ_Contact(in1 := "Dados_Ciclo".POS_EVS_FILT_2, in2 := 'FECHO')
      wire#w4
      { S7_Templates := "SrcType := Int" } EQ_Contact(in1 := "Dados_Ciclo".ETAPA_ANTERIOR, in2 := 5)
   END_RUNG wire#w2
   RUNG wire#w3
      { S7_Templates := "SrcType := String" } EQ_Contact(in1 := "Dados_Ciclo".POS_EVS_FILT_2, in2 := 'LAVAGEM')
      { S7_Templates := "SrcType := String" } EQ_Contact(in1 := "Dados_Ciclo".POS_EVS_FILT_1, in2 := 'FECHO')
   END_RUNG wire#w4
   RUNG wire#w2
      R_Coil( "Etapas_Grafcet".ETAPA_4 )
   END_RUNG
   RUNG wire#w2
      R_Coil( "Etapas_Grafcet".ETAPA_15 )
   END_RUNG
   // the same network as SCL:
   IF ("Etapas_Grafcet".ETAPA_4 AND ("T_LAVAGEM".Q OR "Dados_Ciclo".STOP_CICLO)) OR ("Etapas_Grafcet".ETAPA_15 AND "T_POS_EVS".Q AND ((("Dados_Ciclo".POS_EVS_FILT_1 = 'LAVAGEM') AND ("Dados_Ciclo".POS_EVS_FILT_2 = 'FECHO')) OR (("Dados_Ciclo".POS_EVS_FILT_2 = 'LAVAGEM') AND ("Dados_Ciclo".POS_EVS_FILT_1 = 'FECHO'))) AND ("Dados_Ciclo".ETAPA_ANTERIOR = 5)) THEN
       "Etapas_Grafcet".ETAPA_5 := TRUE;
   END_IF;
   #_w1 := ("Etapas_Grafcet".ETAPA_4 AND ("T_LAVAGEM".Q OR "Dados_Ciclo".STOP_CICLO)) OR ("Etapas_Grafcet".ETAPA_15 AND "T_POS_EVS".Q AND ((("Dados_Ciclo".POS_EVS_FILT_1 = 'LAVAGEM') AND ("Dados_Ciclo".POS_EVS_FILT_2 = 'FECHO')) OR (("Dados_Ciclo".POS_EVS_FILT_2 = 'LAVAGEM') AND ("Dados_Ciclo".POS_EVS_FILT_1 = 'FECHO'))) AND ("Dados_Ciclo".ETAPA_ANTERIOR = 5));
   IF #_w1 THEN
       "Etapas_Grafcet".ETAPA_4 := FALSE;
       "Etapas_Grafcet".ETAPA_15 := FALSE;
   END_IF;
END_REGION

REGION Network 6: Etapa 6 (Passagem à posição de rinse)
   RUNG wire#powerrail
      Contact( "Etapas_Grafcet".ETAPA_5 )
      Contact( "T_STOP_BOMBAS".Q )
      I_Contact( "Dados_Ciclo".STOP_CICLO )
      wire#w1
      S_Coil( "Etapas_Grafcet".ETAPA_6 )
   END_RUNG
   RUNG wire#powerrail
      Contact( "Etapas_Grafcet".ETAPA_11 )
      Contact( "Inputs_HMI".REARME )
   END_RUNG wire#w1
   RUNG wire#powerrail
      Contact( "Etapas_Grafcet".ETAPA_15 )
      Contact( "T_POS_EVS".Q )
      wire#w2
      { S7_Templates := "SrcType := String" } EQ_Contact(in1 := "Dados_Ciclo".POS_EVS_FILT_1, in2 := 'RINSE')
      { S7_Templates := "SrcType := String" } EQ_Contact(in1 := "Dados_Ciclo".POS_EVS_FILT_2, in2 := 'FECHO')
      wire#w3
      { S7_Templates := "SrcType := Int" } EQ_Contact(in1 := "Dados_Ciclo".ETAPA_ANTERIOR, in2 := 6)
   END_RUNG wire#w1
   RUNG wire#w2
      { S7_Templates := "SrcType := String" } EQ_Contact(in1 := "Dados_Ciclo".POS_EVS_FILT_2, in2 := 'RINSE')
      { S7_Templates := "SrcType := String" } EQ_Contact(in1 := "Dados_Ciclo".POS_EVS_FILT_1, in2 := 'FECHO')
   END_RUNG wire#w3
   RUNG wire#w1
      R_Coil( "Etapas_Grafcet".ETAPA_5 )
   END_RUNG
   RUNG wire#w1
      R_Coil( "Etapas_Grafcet".ETAPA_11 )
   END_RUNG
   RUNG wire#w1
      R_Coil( "Etapas_Grafcet".ETAPA_15 )
   END_RUNG
   // the same network as SCL:
   IF ("Etapas_Grafcet".ETAPA_5 AND "T_STOP_BOMBAS".Q AND NOT "Dados_Ciclo".STOP_CICLO) OR ("Etapas_Grafcet".ETAPA_11 AND "Inputs_HMI".REARME) OR ("Etapas_Grafcet".ETAPA_15 AND "T_POS_EVS".Q AND ((("Dados_Ciclo".POS_EVS_FILT_1 = 'RINSE') AND ("Dados_Ciclo".POS_EVS_FILT_2 = 'FECHO')) OR (("Dados_Ciclo".POS_EVS_FILT_2 = 'RINSE') AND ("Dados_Ciclo".POS_EVS_FILT_1 = 'FECHO'))) AND ("Dados_Ciclo".ETAPA_ANTERIOR = 6)) THEN
       "Etapas_Grafcet".ETAPA_6 := TRUE;
   END_IF;
   #_w1 := ("Etapas_Grafcet".ETAPA_5 AND "T_STOP_BOMBAS".Q AND NOT "Dados_Ciclo".STOP_CICLO) OR ("Etapas_Grafcet".ETAPA_11 AND "Inputs_HMI".REARME) OR ("Etapas_Grafcet".ETAPA_15 AND "T_POS_EVS".Q AND ((("Dados_Ciclo".POS_EVS_FILT_1 = 'RINSE') AND ("Dados_Ciclo".POS_EVS_FILT_2 = 'FECHO')) OR (("Dados_Ciclo".POS_EVS_FILT_2 = 'RINSE') AND ("Dados_Ciclo".POS_EVS_FILT_1 = 'FECHO'))) AND ("Dados_Ciclo".ETAPA_ANTERIOR = 6));
   IF #_w1 THEN
       "Etapas_Grafcet".ETAPA_5 := FALSE;
       "Etapas_Grafcet".ETAPA_11 := FALSE;
       "Etapas_Grafcet".ETAPA_15 := FALSE;
   END_IF;
END_REGION

REGION Network 7: Etapa 7 (Em rinse, B1 ligada)
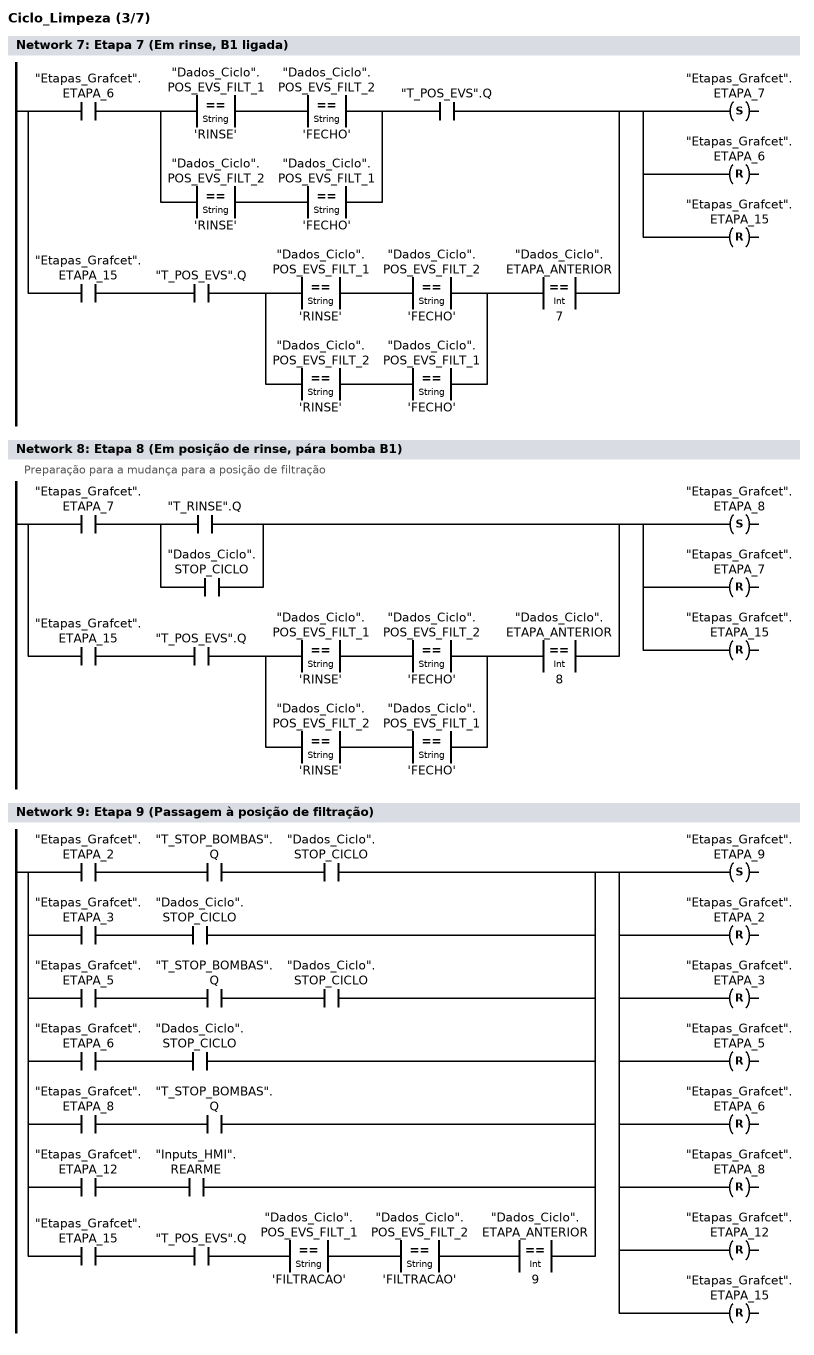
   RUNG wire#powerrail
      Contact( "Etapas_Grafcet".ETAPA_6 )
      wire#w1
      { S7_Templates := "SrcType := String" } EQ_Contact(in1 := "Dados_Ciclo".POS_EVS_FILT_1, in2 := 'RINSE')
      { S7_Templates := "SrcType := String" } EQ_Contact(in1 := "Dados_Ciclo".POS_EVS_FILT_2, in2 := 'FECHO')
      wire#w2
      Contact( "T_POS_EVS".Q )
      wire#w3
      S_Coil( "Etapas_Grafcet".ETAPA_7 )
   END_RUNG
   RUNG wire#w1
      { S7_Templates := "SrcType := String" } EQ_Contact(in1 := "Dados_Ciclo".POS_EVS_FILT_2, in2 := 'RINSE')
      { S7_Templates := "SrcType := String" } EQ_Contact(in1 := "Dados_Ciclo".POS_EVS_FILT_1, in2 := 'FECHO')
   END_RUNG wire#w2
   RUNG wire#powerrail
      Contact( "Etapas_Grafcet".ETAPA_15 )
      Contact( "T_POS_EVS".Q )
      wire#w4
      { S7_Templates := "SrcType := String" } EQ_Contact(in1 := "Dados_Ciclo".POS_EVS_FILT_1, in2 := 'RINSE')
      { S7_Templates := "SrcType := String" } EQ_Contact(in1 := "Dados_Ciclo".POS_EVS_FILT_2, in2 := 'FECHO')
      wire#w5
      { S7_Templates := "SrcType := Int" } EQ_Contact(in1 := "Dados_Ciclo".ETAPA_ANTERIOR, in2 := 7)
   END_RUNG wire#w3
   RUNG wire#w4
      { S7_Templates := "SrcType := String" } EQ_Contact(in1 := "Dados_Ciclo".POS_EVS_FILT_2, in2 := 'RINSE')
      { S7_Templates := "SrcType := String" } EQ_Contact(in1 := "Dados_Ciclo".POS_EVS_FILT_1, in2 := 'FECHO')
   END_RUNG wire#w5
   RUNG wire#w3
      R_Coil( "Etapas_Grafcet".ETAPA_6 )
   END_RUNG
   RUNG wire#w3
      R_Coil( "Etapas_Grafcet".ETAPA_15 )
   END_RUNG
   // the same network as SCL:
   IF ("Etapas_Grafcet".ETAPA_6 AND ((("Dados_Ciclo".POS_EVS_FILT_1 = 'RINSE') AND ("Dados_Ciclo".POS_EVS_FILT_2 = 'FECHO')) OR (("Dados_Ciclo".POS_EVS_FILT_2 = 'RINSE') AND ("Dados_Ciclo".POS_EVS_FILT_1 = 'FECHO'))) AND "T_POS_EVS".Q) OR ("Etapas_Grafcet".ETAPA_15 AND "T_POS_EVS".Q AND ((("Dados_Ciclo".POS_EVS_FILT_1 = 'RINSE') AND ("Dados_Ciclo".POS_EVS_FILT_2 = 'FECHO')) OR (("Dados_Ciclo".POS_EVS_FILT_2 = 'RINSE') AND ("Dados_Ciclo".POS_EVS_FILT_1 = 'FECHO'))) AND ("Dados_Ciclo".ETAPA_ANTERIOR = 7)) THEN
       "Etapas_Grafcet".ETAPA_7 := TRUE;
   END_IF;
   #_w1 := ("Etapas_Grafcet".ETAPA_6 AND ((("Dados_Ciclo".POS_EVS_FILT_1 = 'RINSE') AND ("Dados_Ciclo".POS_EVS_FILT_2 = 'FECHO')) OR (("Dados_Ciclo".POS_EVS_FILT_2 = 'RINSE') AND ("Dados_Ciclo".POS_EVS_FILT_1 = 'FECHO'))) AND "T_POS_EVS".Q) OR ("Etapas_Grafcet".ETAPA_15 AND "T_POS_EVS".Q AND ((("Dados_Ciclo".POS_EVS_FILT_1 = 'RINSE') AND ("Dados_Ciclo".POS_EVS_FILT_2 = 'FECHO')) OR (("Dados_Ciclo".POS_EVS_FILT_2 = 'RINSE') AND ("Dados_Ciclo".POS_EVS_FILT_1 = 'FECHO'))) AND ("Dados_Ciclo".ETAPA_ANTERIOR = 7));
   IF #_w1 THEN
       "Etapas_Grafcet".ETAPA_6 := FALSE;
       "Etapas_Grafcet".ETAPA_15 := FALSE;
   END_IF;
END_REGION

REGION Network 8: Etapa 8 (Em posição de rinse, pára bomba B1)
   // Preparação para a mudança para a posição de filtração
   RUNG wire#powerrail
      Contact( "Etapas_Grafcet".ETAPA_7 )
      wire#w1
      Contact( "T_RINSE".Q )
      wire#w2
      S_Coil( "Etapas_Grafcet".ETAPA_8 )
   END_RUNG
   RUNG wire#w1
      Contact( "Dados_Ciclo".STOP_CICLO )
   END_RUNG wire#w2
   RUNG wire#powerrail
      Contact( "Etapas_Grafcet".ETAPA_15 )
      Contact( "T_POS_EVS".Q )
      wire#w3
      { S7_Templates := "SrcType := String" } EQ_Contact(in1 := "Dados_Ciclo".POS_EVS_FILT_1, in2 := 'RINSE')
      { S7_Templates := "SrcType := String" } EQ_Contact(in1 := "Dados_Ciclo".POS_EVS_FILT_2, in2 := 'FECHO')
      wire#w4
      { S7_Templates := "SrcType := Int" } EQ_Contact(in1 := "Dados_Ciclo".ETAPA_ANTERIOR, in2 := 8)
   END_RUNG wire#w2
   RUNG wire#w3
      { S7_Templates := "SrcType := String" } EQ_Contact(in1 := "Dados_Ciclo".POS_EVS_FILT_2, in2 := 'RINSE')
      { S7_Templates := "SrcType := String" } EQ_Contact(in1 := "Dados_Ciclo".POS_EVS_FILT_1, in2 := 'FECHO')
   END_RUNG wire#w4
   RUNG wire#w2
      R_Coil( "Etapas_Grafcet".ETAPA_7 )
   END_RUNG
   RUNG wire#w2
      R_Coil( "Etapas_Grafcet".ETAPA_15 )
   END_RUNG
   // the same network as SCL:
   IF ("Etapas_Grafcet".ETAPA_7 AND ("T_RINSE".Q OR "Dados_Ciclo".STOP_CICLO)) OR ("Etapas_Grafcet".ETAPA_15 AND "T_POS_EVS".Q AND ((("Dados_Ciclo".POS_EVS_FILT_1 = 'RINSE') AND ("Dados_Ciclo".POS_EVS_FILT_2 = 'FECHO')) OR (("Dados_Ciclo".POS_EVS_FILT_2 = 'RINSE') AND ("Dados_Ciclo".POS_EVS_FILT_1 = 'FECHO'))) AND ("Dados_Ciclo".ETAPA_ANTERIOR = 8)) THEN
       "Etapas_Grafcet".ETAPA_8 := TRUE;
   END_IF;
   #_w1 := ("Etapas_Grafcet".ETAPA_7 AND ("T_RINSE".Q OR "Dados_Ciclo".STOP_CICLO)) OR ("Etapas_Grafcet".ETAPA_15 AND "T_POS_EVS".Q AND ((("Dados_Ciclo".POS_EVS_FILT_1 = 'RINSE') AND ("Dados_Ciclo".POS_EVS_FILT_2 = 'FECHO')) OR (("Dados_Ciclo".POS_EVS_FILT_2 = 'RINSE') AND ("Dados_Ciclo".POS_EVS_FILT_1 = 'FECHO'))) AND ("Dados_Ciclo".ETAPA_ANTERIOR = 8));
   IF #_w1 THEN
       "Etapas_Grafcet".ETAPA_7 := FALSE;
       "Etapas_Grafcet".ETAPA_15 := FALSE;
   END_IF;
END_REGION

REGION Network 9: Etapa 9 (Passagem à posição de filtração)
   RUNG wire#powerrail
      Contact( "Etapas_Grafcet".ETAPA_2 )
      Contact( "T_STOP_BOMBAS".Q )
      Contact( "Dados_Ciclo".STOP_CICLO )
      wire#w1
      S_Coil( "Etapas_Grafcet".ETAPA_9 )
   END_RUNG
   RUNG wire#powerrail
      Contact( "Etapas_Grafcet".ETAPA_3 )
      Contact( "Dados_Ciclo".STOP_CICLO )
   END_RUNG wire#w1
   RUNG wire#powerrail
      Contact( "Etapas_Grafcet".ETAPA_5 )
      Contact( "T_STOP_BOMBAS".Q )
      Contact( "Dados_Ciclo".STOP_CICLO )
   END_RUNG wire#w1
   RUNG wire#powerrail
      Contact( "Etapas_Grafcet".ETAPA_6 )
      Contact( "Dados_Ciclo".STOP_CICLO )
   END_RUNG wire#w1
   RUNG wire#powerrail
      Contact( "Etapas_Grafcet".ETAPA_8 )
      Contact( "T_STOP_BOMBAS".Q )
   END_RUNG wire#w1
   RUNG wire#powerrail
      Contact( "Etapas_Grafcet".ETAPA_12 )
      Contact( "Inputs_HMI".REARME )
   END_RUNG wire#w1
   RUNG wire#powerrail
      Contact( "Etapas_Grafcet".ETAPA_15 )
      Contact( "T_POS_EVS".Q )
      { S7_Templates := "SrcType := String" } EQ_Contact(in1 := "Dados_Ciclo".POS_EVS_FILT_1, in2 := 'FILTRACAO')
      { S7_Templates := "SrcType := String" } EQ_Contact(in1 := "Dados_Ciclo".POS_EVS_FILT_2, in2 := 'FILTRACAO')
      { S7_Templates := "SrcType := Int" } EQ_Contact(in1 := "Dados_Ciclo".ETAPA_ANTERIOR, in2 := 9)
   END_RUNG wire#w1
   RUNG wire#w1
      R_Coil( "Etapas_Grafcet".ETAPA_2 )
   END_RUNG
   RUNG wire#w1
      R_Coil( "Etapas_Grafcet".ETAPA_3 )
   END_RUNG
   RUNG wire#w1
      R_Coil( "Etapas_Grafcet".ETAPA_5 )
   END_RUNG
   RUNG wire#w1
      R_Coil( "Etapas_Grafcet".ETAPA_6 )
   END_RUNG
   RUNG wire#w1
      R_Coil( "Etapas_Grafcet".ETAPA_8 )
   END_RUNG
   RUNG wire#w1
      R_Coil( "Etapas_Grafcet".ETAPA_12 )
   END_RUNG
   RUNG wire#w1
      R_Coil( "Etapas_Grafcet".ETAPA_15 )
   END_RUNG
   // the same network as SCL:
   IF ("Etapas_Grafcet".ETAPA_2 AND "T_STOP_BOMBAS".Q AND "Dados_Ciclo".STOP_CICLO) OR ("Etapas_Grafcet".ETAPA_3 AND "Dados_Ciclo".STOP_CICLO) OR ("Etapas_Grafcet".ETAPA_5 AND "T_STOP_BOMBAS".Q AND "Dados_Ciclo".STOP_CICLO) OR ("Etapas_Grafcet".ETAPA_6 AND "Dados_Ciclo".STOP_CICLO) OR ("Etapas_Grafcet".ETAPA_8 AND "T_STOP_BOMBAS".Q) OR ("Etapas_Grafcet".ETAPA_12 AND "Inputs_HMI".REARME) OR ("Etapas_Grafcet".ETAPA_15 AND "T_POS_EVS".Q AND ("Dados_Ciclo".POS_EVS_FILT_1 = 'FILTRACAO') AND ("Dados_Ciclo".POS_EVS_FILT_2 = 'FILTRACAO') AND ("Dados_Ciclo".ETAPA_ANTERIOR = 9)) THEN
       "Etapas_Grafcet".ETAPA_9 := TRUE;
   END_IF;
   #_w1 := ("Etapas_Grafcet".ETAPA_2 AND "T_STOP_BOMBAS".Q AND "Dados_Ciclo".STOP_CICLO) OR ("Etapas_Grafcet".ETAPA_3 AND "Dados_Ciclo".STOP_CICLO) OR ("Etapas_Grafcet".ETAPA_5 AND "T_STOP_BOMBAS".Q AND "Dados_Ciclo".STOP_CICLO) OR ("Etapas_Grafcet".ETAPA_6 AND "Dados_Ciclo".STOP_CICLO) OR ("Etapas_Grafcet".ETAPA_8 AND "T_STOP_BOMBAS".Q) OR ("Etapas_Grafcet".ETAPA_12 AND "Inputs_HMI".REARME) OR ("Etapas_Grafcet".ETAPA_15 AND "T_POS_EVS".Q AND ("Dados_Ciclo".POS_EVS_FILT_1 = 'FILTRACAO') AND ("Dados_Ciclo".POS_EVS_FILT_2 = 'FILTRACAO') AND ("Dados_Ciclo".ETAPA_ANTERIOR = 9));
   IF #_w1 THEN
       "Etapas_Grafcet".ETAPA_2 := FALSE;
       "Etapas_Grafcet".ETAPA_3 := FALSE;
       "Etapas_Grafcet".ETAPA_5 := FALSE;
       "Etapas_Grafcet".ETAPA_6 := FALSE;
       "Etapas_Grafcet".ETAPA_8 := FALSE;
       "Etapas_Grafcet".ETAPA_12 := FALSE;
       "Etapas_Grafcet".ETAPA_15 := FALSE;
   END_IF;
END_REGION

REGION Network 10: ETAPA 10 (Alarme posição lavagem)
   // As ev's não estão na posição de lavagem / fecho
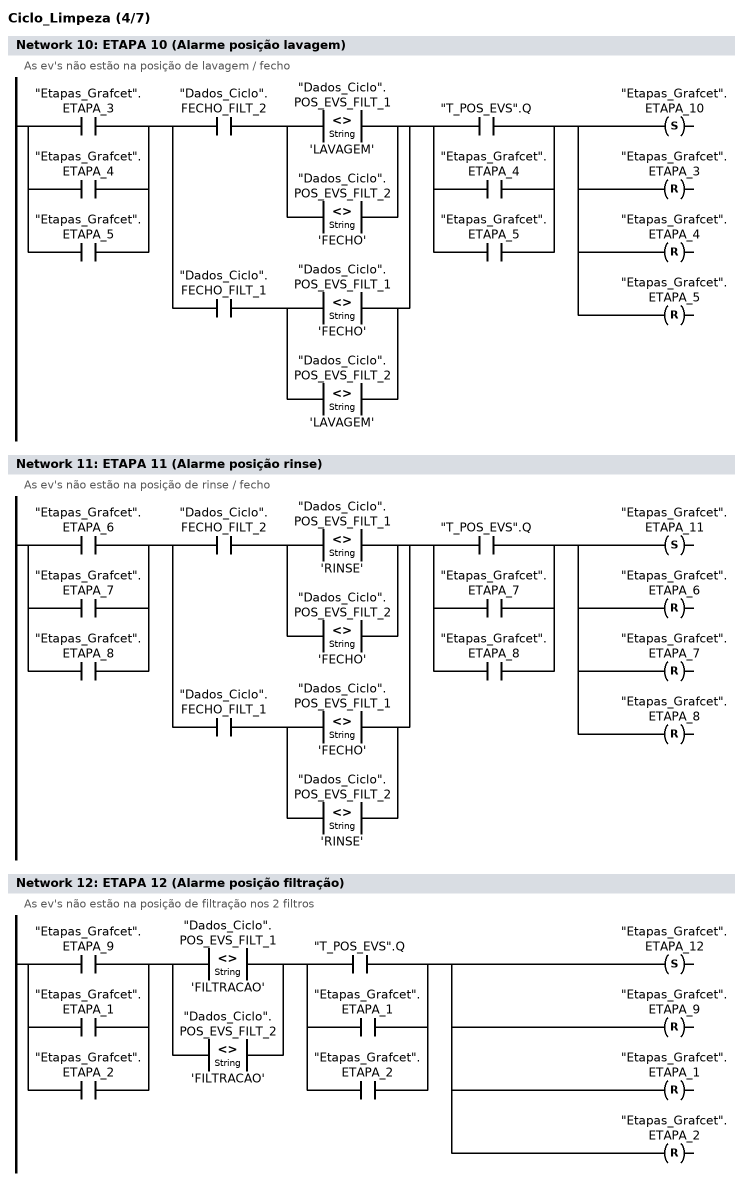
   RUNG wire#powerrail
      Contact( "Etapas_Grafcet".ETAPA_3 )
      wire#w1
      Contact( "Dados_Ciclo".FECHO_FILT_2 )
      wire#w2
      { S7_Templates := "SrcType := String" } NE_Contact(in1 := "Dados_Ciclo".POS_EVS_FILT_1, in2 := 'LAVAGEM')
      wire#w3
      Contact( "T_POS_EVS".Q )
      wire#w5
      S_Coil( "Etapas_Grafcet".ETAPA_10 )
   END_RUNG
   RUNG wire#powerrail
      Contact( "Etapas_Grafcet".ETAPA_4 )
   END_RUNG wire#w1
   RUNG wire#powerrail
      Contact( "Etapas_Grafcet".ETAPA_5 )
   END_RUNG wire#w1
   RUNG wire#w2
      { S7_Templates := "SrcType := String" } NE_Contact(in1 := "Dados_Ciclo".POS_EVS_FILT_2, in2 := 'FECHO')
   END_RUNG wire#w3
   RUNG wire#w1
      Contact( "Dados_Ciclo".FECHO_FILT_1 )
      wire#w4
      { S7_Templates := "SrcType := String" } NE_Contact(in1 := "Dados_Ciclo".POS_EVS_FILT_1, in2 := 'FECHO')
   END_RUNG wire#w3
   RUNG wire#w4
      { S7_Templates := "SrcType := String" } NE_Contact(in1 := "Dados_Ciclo".POS_EVS_FILT_2, in2 := 'LAVAGEM')
   END_RUNG wire#w3
   RUNG wire#w3
      Contact( "Etapas_Grafcet".ETAPA_4 )
   END_RUNG wire#w5
   RUNG wire#w3
      Contact( "Etapas_Grafcet".ETAPA_5 )
   END_RUNG wire#w5
   RUNG wire#w5
      R_Coil( "Etapas_Grafcet".ETAPA_3 )
   END_RUNG
   RUNG wire#w5
      R_Coil( "Etapas_Grafcet".ETAPA_4 )
   END_RUNG
   RUNG wire#w5
      R_Coil( "Etapas_Grafcet".ETAPA_5 )
   END_RUNG
   // the same network as SCL:
   IF ("Etapas_Grafcet".ETAPA_3 OR "Etapas_Grafcet".ETAPA_4 OR "Etapas_Grafcet".ETAPA_5) AND (("Dados_Ciclo".FECHO_FILT_2 AND (("Dados_Ciclo".POS_EVS_FILT_1 <> 'LAVAGEM') OR ("Dados_Ciclo".POS_EVS_FILT_2 <> 'FECHO'))) OR ("Dados_Ciclo".FECHO_FILT_1 AND (("Dados_Ciclo".POS_EVS_FILT_1 <> 'FECHO') OR ("Dados_Ciclo".POS_EVS_FILT_2 <> 'LAVAGEM')))) AND ("T_POS_EVS".Q OR "Etapas_Grafcet".ETAPA_4 OR "Etapas_Grafcet".ETAPA_5) THEN
       "Etapas_Grafcet".ETAPA_10 := TRUE;
   END_IF;
   #_w1 := ("Etapas_Grafcet".ETAPA_3 OR "Etapas_Grafcet".ETAPA_4 OR "Etapas_Grafcet".ETAPA_5) AND (("Dados_Ciclo".FECHO_FILT_2 AND (("Dados_Ciclo".POS_EVS_FILT_1 <> 'LAVAGEM') OR ("Dados_Ciclo".POS_EVS_FILT_2 <> 'FECHO'))) OR ("Dados_Ciclo".FECHO_FILT_1 AND (("Dados_Ciclo".POS_EVS_FILT_1 <> 'FECHO') OR ("Dados_Ciclo".POS_EVS_FILT_2 <> 'LAVAGEM')))) AND ("T_POS_EVS".Q OR "Etapas_Grafcet".ETAPA_4 OR "Etapas_Grafcet".ETAPA_5);
   IF #_w1 THEN
       "Etapas_Grafcet".ETAPA_3 := FALSE;
       "Etapas_Grafcet".ETAPA_4 := FALSE;
       "Etapas_Grafcet".ETAPA_5 := FALSE;
   END_IF;
END_REGION

REGION Network 11: ETAPA 11 (Alarme posição rinse)
   // As ev's não estão na posição de rinse / fecho
   RUNG wire#powerrail
      Contact( "Etapas_Grafcet".ETAPA_6 )
      wire#w1
      Contact( "Dados_Ciclo".FECHO_FILT_2 )
      wire#w2
      { S7_Templates := "SrcType := String" } NE_Contact(in1 := "Dados_Ciclo".POS_EVS_FILT_1, in2 := 'RINSE')
      wire#w3
      Contact( "T_POS_EVS".Q )
      wire#w5
      S_Coil( "Etapas_Grafcet".ETAPA_11 )
   END_RUNG
   RUNG wire#powerrail
      Contact( "Etapas_Grafcet".ETAPA_7 )
   END_RUNG wire#w1
   RUNG wire#powerrail
      Contact( "Etapas_Grafcet".ETAPA_8 )
   END_RUNG wire#w1
   RUNG wire#w2
      { S7_Templates := "SrcType := String" } NE_Contact(in1 := "Dados_Ciclo".POS_EVS_FILT_2, in2 := 'FECHO')
   END_RUNG wire#w3
   RUNG wire#w1
      Contact( "Dados_Ciclo".FECHO_FILT_1 )
      wire#w4
      { S7_Templates := "SrcType := String" } NE_Contact(in1 := "Dados_Ciclo".POS_EVS_FILT_1, in2 := 'FECHO')
   END_RUNG wire#w3
   RUNG wire#w4
      { S7_Templates := "SrcType := String" } NE_Contact(in1 := "Dados_Ciclo".POS_EVS_FILT_2, in2 := 'RINSE')
   END_RUNG wire#w3
   RUNG wire#w3
      Contact( "Etapas_Grafcet".ETAPA_7 )
   END_RUNG wire#w5
   RUNG wire#w3
      Contact( "Etapas_Grafcet".ETAPA_8 )
   END_RUNG wire#w5
   RUNG wire#w5
      R_Coil( "Etapas_Grafcet".ETAPA_6 )
   END_RUNG
   RUNG wire#w5
      R_Coil( "Etapas_Grafcet".ETAPA_7 )
   END_RUNG
   RUNG wire#w5
      R_Coil( "Etapas_Grafcet".ETAPA_8 )
   END_RUNG
   // the same network as SCL:
   IF ("Etapas_Grafcet".ETAPA_6 OR "Etapas_Grafcet".ETAPA_7 OR "Etapas_Grafcet".ETAPA_8) AND (("Dados_Ciclo".FECHO_FILT_2 AND (("Dados_Ciclo".POS_EVS_FILT_1 <> 'RINSE') OR ("Dados_Ciclo".POS_EVS_FILT_2 <> 'FECHO'))) OR ("Dados_Ciclo".FECHO_FILT_1 AND (("Dados_Ciclo".POS_EVS_FILT_1 <> 'FECHO') OR ("Dados_Ciclo".POS_EVS_FILT_2 <> 'RINSE')))) AND ("T_POS_EVS".Q OR "Etapas_Grafcet".ETAPA_7 OR "Etapas_Grafcet".ETAPA_8) THEN
       "Etapas_Grafcet".ETAPA_11 := TRUE;
   END_IF;
   #_w1 := ("Etapas_Grafcet".ETAPA_6 OR "Etapas_Grafcet".ETAPA_7 OR "Etapas_Grafcet".ETAPA_8) AND (("Dados_Ciclo".FECHO_FILT_2 AND (("Dados_Ciclo".POS_EVS_FILT_1 <> 'RINSE') OR ("Dados_Ciclo".POS_EVS_FILT_2 <> 'FECHO'))) OR ("Dados_Ciclo".FECHO_FILT_1 AND (("Dados_Ciclo".POS_EVS_FILT_1 <> 'FECHO') OR ("Dados_Ciclo".POS_EVS_FILT_2 <> 'RINSE')))) AND ("T_POS_EVS".Q OR "Etapas_Grafcet".ETAPA_7 OR "Etapas_Grafcet".ETAPA_8);
   IF #_w1 THEN
       "Etapas_Grafcet".ETAPA_6 := FALSE;
       "Etapas_Grafcet".ETAPA_7 := FALSE;
       "Etapas_Grafcet".ETAPA_8 := FALSE;
   END_IF;
END_REGION

REGION Network 12: ETAPA 12 (Alarme posição filtração)
   // As ev's não estão na posição de filtração nos 2 filtros
   RUNG wire#powerrail
      Contact( "Etapas_Grafcet".ETAPA_9 )
      wire#w1
      { S7_Templates := "SrcType := String" } NE_Contact(in1 := "Dados_Ciclo".POS_EVS_FILT_1, in2 := 'FILTRACAO')
      wire#w2
      Contact( "T_POS_EVS".Q )
      wire#w3
      S_Coil( "Etapas_Grafcet".ETAPA_12 )
   END_RUNG
   RUNG wire#powerrail
      Contact( "Etapas_Grafcet".ETAPA_1 )
   END_RUNG wire#w1
   RUNG wire#powerrail
      Contact( "Etapas_Grafcet".ETAPA_2 )
   END_RUNG wire#w1
   RUNG wire#w1
      { S7_Templates := "SrcType := String" } NE_Contact(in1 := "Dados_Ciclo".POS_EVS_FILT_2, in2 := 'FILTRACAO')
   END_RUNG wire#w2
   RUNG wire#w2
      Contact( "Etapas_Grafcet".ETAPA_1 )
   END_RUNG wire#w3
   RUNG wire#w2
      Contact( "Etapas_Grafcet".ETAPA_2 )
   END_RUNG wire#w3
   RUNG wire#w3
      R_Coil( "Etapas_Grafcet".ETAPA_9 )
   END_RUNG
   RUNG wire#w3
      R_Coil( "Etapas_Grafcet".ETAPA_1 )
   END_RUNG
   RUNG wire#w3
      R_Coil( "Etapas_Grafcet".ETAPA_2 )
   END_RUNG
   // the same network as SCL:
   IF ("Etapas_Grafcet".ETAPA_9 OR "Etapas_Grafcet".ETAPA_1 OR "Etapas_Grafcet".ETAPA_2) AND (("Dados_Ciclo".POS_EVS_FILT_1 <> 'FILTRACAO') OR ("Dados_Ciclo".POS_EVS_FILT_2 <> 'FILTRACAO')) AND ("T_POS_EVS".Q OR "Etapas_Grafcet".ETAPA_1 OR "Etapas_Grafcet".ETAPA_2) THEN
       "Etapas_Grafcet".ETAPA_12 := TRUE;
   END_IF;
   #_w1 := ("Etapas_Grafcet".ETAPA_9 OR "Etapas_Grafcet".ETAPA_1 OR "Etapas_Grafcet".ETAPA_2) AND (("Dados_Ciclo".POS_EVS_FILT_1 <> 'FILTRACAO') OR ("Dados_Ciclo".POS_EVS_FILT_2 <> 'FILTRACAO')) AND ("T_POS_EVS".Q OR "Etapas_Grafcet".ETAPA_1 OR "Etapas_Grafcet".ETAPA_2);
   IF #_w1 THEN
       "Etapas_Grafcet".ETAPA_9 := FALSE;
       "Etapas_Grafcet".ETAPA_1 := FALSE;
       "Etapas_Grafcet".ETAPA_2 := FALSE;
   END_IF;
END_REGION

REGION Network 13: Etapa 13 (Preparação para modo manual)
   // A etapa_n são as etapas de 1 a 9. A etapa 13 corresponde à preparação para entrada em manual. Param as bombas e mantém a posição das válvulas da etapa anterior. O reset às etapas de 1 a 9 é feito em Controlo_Ciclo_Manual
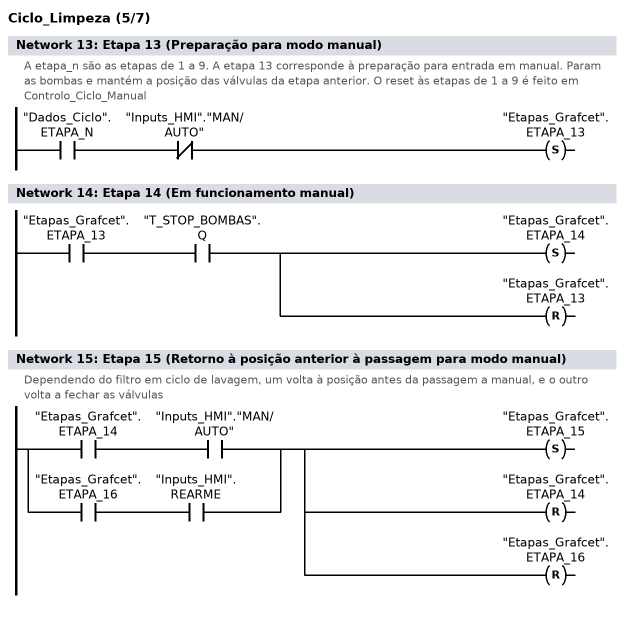
   RUNG wire#powerrail
      Contact( "Dados_Ciclo".ETAPA_N )
      I_Contact( "Inputs_HMI"."MAN/AUTO" )
      S_Coil( "Etapas_Grafcet".ETAPA_13 )
   END_RUNG
   // the same network as SCL:
   IF "Dados_Ciclo".ETAPA_N AND NOT "Inputs_HMI"."MAN/AUTO" THEN "Etapas_Grafcet".ETAPA_13 := TRUE; END_IF;
END_REGION

REGION Network 14: Etapa 14 (Em funcionamento manual)
   RUNG wire#powerrail
      Contact( "Etapas_Grafcet".ETAPA_13 )
      Contact( "T_STOP_BOMBAS".Q )
      wire#w1
      S_Coil( "Etapas_Grafcet".ETAPA_14 )
   END_RUNG
   RUNG wire#w1
      R_Coil( "Etapas_Grafcet".ETAPA_13 )
   END_RUNG
   // the same network as SCL:
   IF "Etapas_Grafcet".ETAPA_13 AND "T_STOP_BOMBAS".Q THEN
       "Etapas_Grafcet".ETAPA_14 := TRUE;
       "Etapas_Grafcet".ETAPA_13 := FALSE;
   END_IF;
END_REGION

REGION Network 15: Etapa 15 (Retorno à posição anterior à passagem para modo manual)
   // Dependendo do filtro em ciclo de lavagem, um volta à posição antes da passagem a manual, e o outro volta a fechar as válvulas
   RUNG wire#powerrail
      Contact( "Etapas_Grafcet".ETAPA_14 )
      Contact( "Inputs_HMI"."MAN/AUTO" )
      wire#w1
      S_Coil( "Etapas_Grafcet".ETAPA_15 )
   END_RUNG
   RUNG wire#powerrail
      Contact( "Etapas_Grafcet".ETAPA_16 )
      Contact( "Inputs_HMI".REARME )
   END_RUNG wire#w1
   RUNG wire#w1
      R_Coil( "Etapas_Grafcet".ETAPA_14 )
   END_RUNG
   RUNG wire#w1
      R_Coil( "Etapas_Grafcet".ETAPA_16 )
   END_RUNG
   // the same network as SCL:
   IF ("Etapas_Grafcet".ETAPA_14 AND "Inputs_HMI"."MAN/AUTO") OR ("Etapas_Grafcet".ETAPA_16 AND "Inputs_HMI".REARME) THEN
       "Etapas_Grafcet".ETAPA_15 := TRUE;
   END_IF;
   #_w1 := ("Etapas_Grafcet".ETAPA_14 AND "Inputs_HMI"."MAN/AUTO") OR ("Etapas_Grafcet".ETAPA_16 AND "Inputs_HMI".REARME);
   IF #_w1 THEN
       "Etapas_Grafcet".ETAPA_14 := FALSE;
       "Etapas_Grafcet".ETAPA_16 := FALSE;
   END_IF;
END_REGION

REGION Network 16: Etapa 16 (alarme em modo manual)
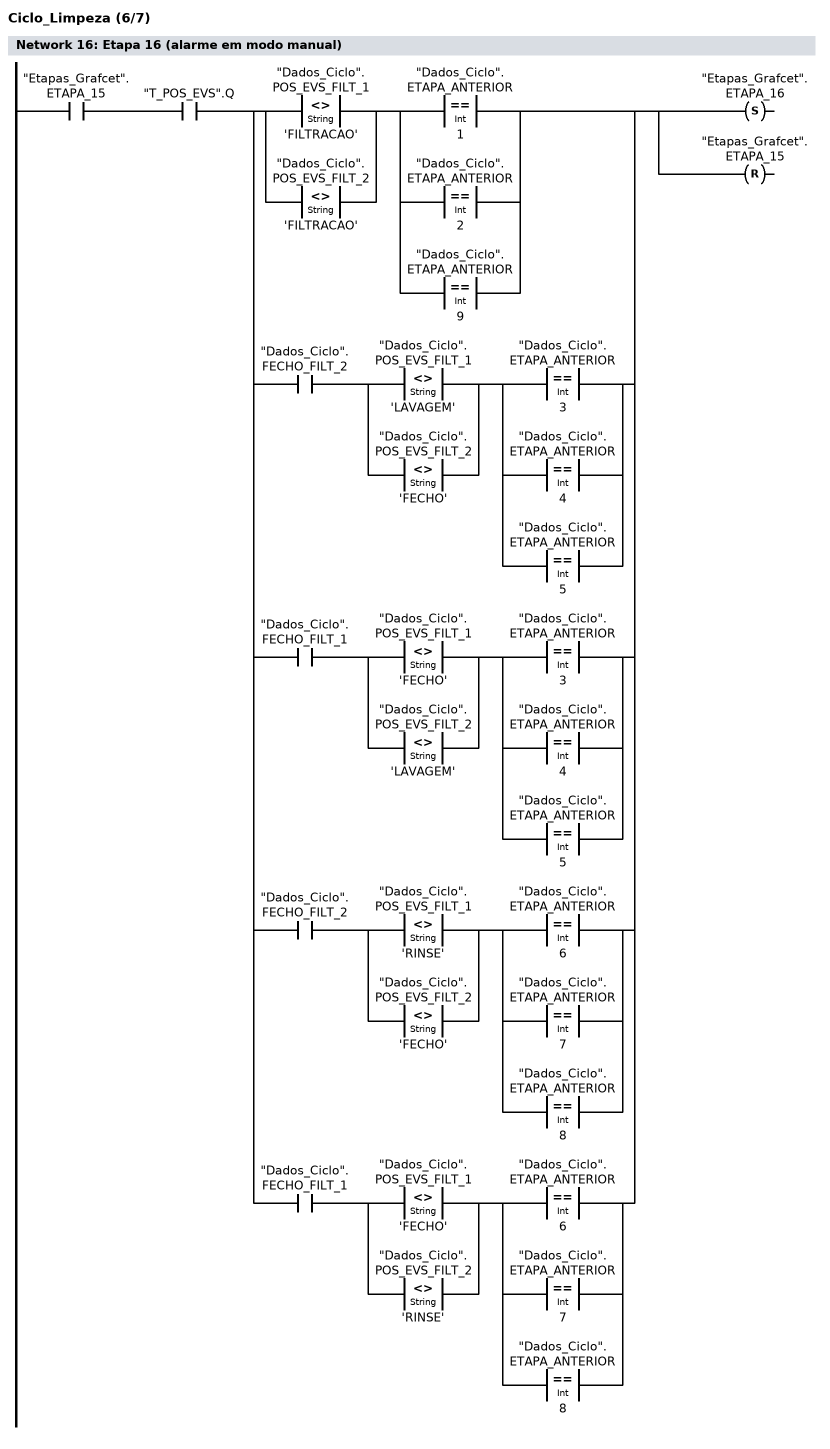
   RUNG wire#powerrail
      Contact( "Etapas_Grafcet".ETAPA_15 )
      Contact( "T_POS_EVS".Q )
      wire#w1
      { S7_Templates := "SrcType := String" } NE_Contact(in1 := "Dados_Ciclo".POS_EVS_FILT_1, in2 := 'FILTRACAO')
      wire#w2
      { S7_Templates := "SrcType := Int" } EQ_Contact(in1 := "Dados_Ciclo".ETAPA_ANTERIOR, in2 := 1)
      wire#w3
      S_Coil( "Etapas_Grafcet".ETAPA_16 )
   END_RUNG
   RUNG wire#w1
      { S7_Templates := "SrcType := String" } NE_Contact(in1 := "Dados_Ciclo".POS_EVS_FILT_2, in2 := 'FILTRACAO')
   END_RUNG wire#w2
   RUNG wire#w2
      { S7_Templates := "SrcType := Int" } EQ_Contact(in1 := "Dados_Ciclo".ETAPA_ANTERIOR, in2 := 2)
   END_RUNG wire#w3
   RUNG wire#w2
      { S7_Templates := "SrcType := Int" } EQ_Contact(in1 := "Dados_Ciclo".ETAPA_ANTERIOR, in2 := 9)
   END_RUNG wire#w3
   RUNG wire#w1
      Contact( "Dados_Ciclo".FECHO_FILT_2 )
      wire#w4
      { S7_Templates := "SrcType := String" } NE_Contact(in1 := "Dados_Ciclo".POS_EVS_FILT_1, in2 := 'LAVAGEM')
      wire#w5
      { S7_Templates := "SrcType := Int" } EQ_Contact(in1 := "Dados_Ciclo".ETAPA_ANTERIOR, in2 := 3)
   END_RUNG wire#w3
   RUNG wire#w4
      { S7_Templates := "SrcType := String" } NE_Contact(in1 := "Dados_Ciclo".POS_EVS_FILT_2, in2 := 'FECHO')
   END_RUNG wire#w5
   RUNG wire#w5
      { S7_Templates := "SrcType := Int" } EQ_Contact(in1 := "Dados_Ciclo".ETAPA_ANTERIOR, in2 := 4)
   END_RUNG wire#w3
   RUNG wire#w5
      { S7_Templates := "SrcType := Int" } EQ_Contact(in1 := "Dados_Ciclo".ETAPA_ANTERIOR, in2 := 5)
   END_RUNG wire#w3
   RUNG wire#w1
      Contact( "Dados_Ciclo".FECHO_FILT_1 )
      wire#w6
      { S7_Templates := "SrcType := String" } NE_Contact(in1 := "Dados_Ciclo".POS_EVS_FILT_1, in2 := 'FECHO')
      wire#w7
      { S7_Templates := "SrcType := Int" } EQ_Contact(in1 := "Dados_Ciclo".ETAPA_ANTERIOR, in2 := 3)
   END_RUNG wire#w3
   RUNG wire#w6
      { S7_Templates := "SrcType := String" } NE_Contact(in1 := "Dados_Ciclo".POS_EVS_FILT_2, in2 := 'LAVAGEM')
   END_RUNG wire#w7
   RUNG wire#w7
      { S7_Templates := "SrcType := Int" } EQ_Contact(in1 := "Dados_Ciclo".ETAPA_ANTERIOR, in2 := 4)
   END_RUNG wire#w3
   RUNG wire#w7
      { S7_Templates := "SrcType := Int" } EQ_Contact(in1 := "Dados_Ciclo".ETAPA_ANTERIOR, in2 := 5)
   END_RUNG wire#w3
   RUNG wire#w1
      Contact( "Dados_Ciclo".FECHO_FILT_2 )
      wire#w8
      { S7_Templates := "SrcType := String" } NE_Contact(in1 := "Dados_Ciclo".POS_EVS_FILT_1, in2 := 'RINSE')
      wire#w9
      { S7_Templates := "SrcType := Int" } EQ_Contact(in1 := "Dados_Ciclo".ETAPA_ANTERIOR, in2 := 6)
   END_RUNG wire#w3
   RUNG wire#w8
      { S7_Templates := "SrcType := String" } NE_Contact(in1 := "Dados_Ciclo".POS_EVS_FILT_2, in2 := 'FECHO')
   END_RUNG wire#w9
   RUNG wire#w9
      { S7_Templates := "SrcType := Int" } EQ_Contact(in1 := "Dados_Ciclo".ETAPA_ANTERIOR, in2 := 7)
   END_RUNG wire#w3
   RUNG wire#w9
      { S7_Templates := "SrcType := Int" } EQ_Contact(in1 := "Dados_Ciclo".ETAPA_ANTERIOR, in2 := 8)
   END_RUNG wire#w3
   RUNG wire#w1
      Contact( "Dados_Ciclo".FECHO_FILT_1 )
      wire#w10
      { S7_Templates := "SrcType := String" } NE_Contact(in1 := "Dados_Ciclo".POS_EVS_FILT_1, in2 := 'FECHO')
      wire#w11
      { S7_Templates := "SrcType := Int" } EQ_Contact(in1 := "Dados_Ciclo".ETAPA_ANTERIOR, in2 := 6)
   END_RUNG wire#w3
   RUNG wire#w10
      { S7_Templates := "SrcType := String" } NE_Contact(in1 := "Dados_Ciclo".POS_EVS_FILT_2, in2 := 'RINSE')
   END_RUNG wire#w11
   RUNG wire#w11
      { S7_Templates := "SrcType := Int" } EQ_Contact(in1 := "Dados_Ciclo".ETAPA_ANTERIOR, in2 := 7)
   END_RUNG wire#w3
   RUNG wire#w11
      { S7_Templates := "SrcType := Int" } EQ_Contact(in1 := "Dados_Ciclo".ETAPA_ANTERIOR, in2 := 8)
   END_RUNG wire#w3
   RUNG wire#w3
      R_Coil( "Etapas_Grafcet".ETAPA_15 )
   END_RUNG
   // the same network as SCL:
   IF "Etapas_Grafcet".ETAPA_15 AND "T_POS_EVS".Q AND (((("Dados_Ciclo".POS_EVS_FILT_1 <> 'FILTRACAO') OR ("Dados_Ciclo".POS_EVS_FILT_2 <> 'FILTRACAO')) AND (("Dados_Ciclo".ETAPA_ANTERIOR = 1) OR ("Dados_Ciclo".ETAPA_ANTERIOR = 2) OR ("Dados_Ciclo".ETAPA_ANTERIOR = 9))) OR ("Dados_Ciclo".FECHO_FILT_2 AND (("Dados_Ciclo".POS_EVS_FILT_1 <> 'LAVAGEM') OR ("Dados_Ciclo".POS_EVS_FILT_2 <> 'FECHO')) AND (("Dados_Ciclo".ETAPA_ANTERIOR = 3) OR ("Dados_Ciclo".ETAPA_ANTERIOR = 4) OR ("Dados_Ciclo".ETAPA_ANTERIOR = 5))) OR ("Dados_Ciclo".FECHO_FILT_1 AND (("Dados_Ciclo".POS_EVS_FILT_1 <> 'FECHO') OR ("Dados_Ciclo".POS_EVS_FILT_2 <> 'LAVAGEM')) AND (("Dados_Ciclo".ETAPA_ANTERIOR = 3) OR ("Dados_Ciclo".ETAPA_ANTERIOR = 4) OR ("Dados_Ciclo".ETAPA_ANTERIOR = 5))) OR ("Dados_Ciclo".FECHO_FILT_2 AND (("Dados_Ciclo".POS_EVS_FILT_1 <> 'RINSE') OR ("Dados_Ciclo".POS_EVS_FILT_2 <> 'FECHO')) AND (("Dados_Ciclo".ETAPA_ANTERIOR = 6) OR ("Dados_Ciclo".ETAPA_ANTERIOR = 7) OR ("Dados_Ciclo".ETAPA_ANTERIOR = 8))) OR ("Dados_Ciclo".FECHO_FILT_1 AND (("Dados_Ciclo".POS_EVS_FILT_1 <> 'FECHO') OR ("Dados_Ciclo".POS_EVS_FILT_2 <> 'RINSE')) AND (("Dados_Ciclo".ETAPA_ANTERIOR = 6) OR ("Dados_Ciclo".ETAPA_ANTERIOR = 7) OR ("Dados_Ciclo".ETAPA_ANTERIOR = 8)))) THEN
       "Etapas_Grafcet".ETAPA_16 := TRUE;
       "Etapas_Grafcet".ETAPA_15 := FALSE;
   END_IF;
END_REGION

REGION Network 17: Tempo de paragem das bombas (T1 no grafcet)
   // Espera um dado tempo para que as bombas parem, de modo a poder mudar a posição das ev's
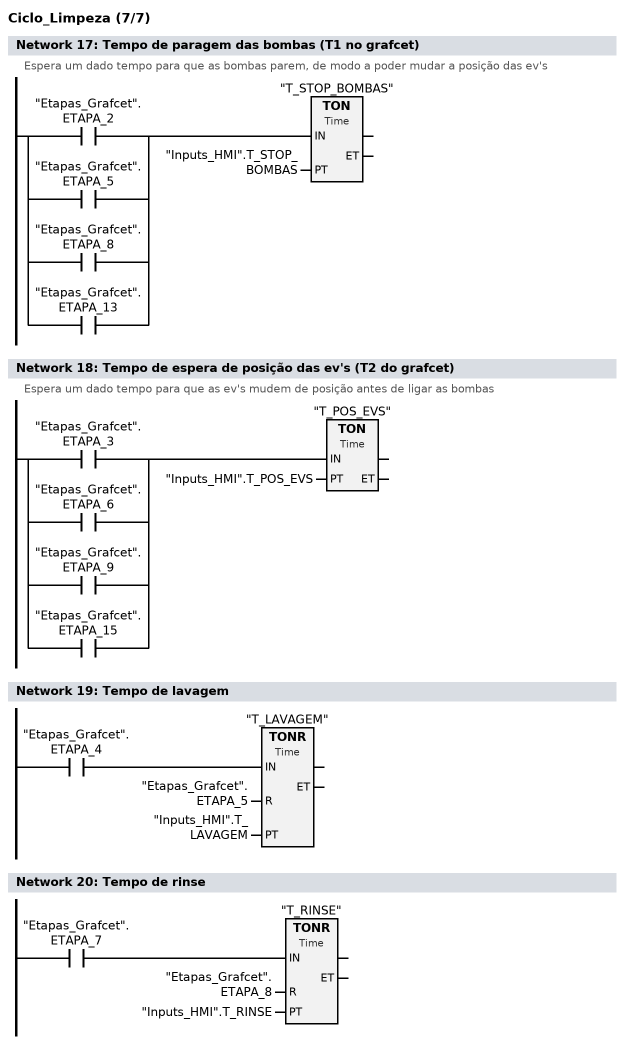
   RUNG wire#powerrail
      Contact( "Etapas_Grafcet".ETAPA_2 )
      wire#w1
      { S7_Templates := "time_type := Time" } "T_STOP_BOMBAS".TON(pt := "Inputs_HMI".T_STOP_BOMBAS, et =>)
   END_RUNG
   RUNG wire#powerrail
      Contact( "Etapas_Grafcet".ETAPA_5 )
   END_RUNG wire#w1
   RUNG wire#powerrail
      Contact( "Etapas_Grafcet".ETAPA_8 )
   END_RUNG wire#w1
   RUNG wire#powerrail
      Contact( "Etapas_Grafcet".ETAPA_13 )
   END_RUNG wire#w1
   // the same network as SCL:
   "T_STOP_BOMBAS".TON(IN := "Etapas_Grafcet".ETAPA_2 OR "Etapas_Grafcet".ETAPA_5 OR "Etapas_Grafcet".ETAPA_8 OR "Etapas_Grafcet".ETAPA_13,
                       PT := "Inputs_HMI".T_STOP_BOMBAS);
END_REGION

REGION Network 18: Tempo de espera de posição das ev's (T2 do grafcet)
   // Espera um dado tempo para que as ev's mudem de posição antes de ligar as bombas
   RUNG wire#powerrail
      Contact( "Etapas_Grafcet".ETAPA_3 )
      wire#w1
      { S7_Templates := "time_type := Time" } "T_POS_EVS".TON(pt := "Inputs_HMI".T_POS_EVS, et =>)
   END_RUNG
   RUNG wire#powerrail
      Contact( "Etapas_Grafcet".ETAPA_6 )
   END_RUNG wire#w1
   RUNG wire#powerrail
      Contact( "Etapas_Grafcet".ETAPA_9 )
   END_RUNG wire#w1
   RUNG wire#powerrail
      Contact( "Etapas_Grafcet".ETAPA_15 )
   END_RUNG wire#w1
   // the same network as SCL:
   "T_POS_EVS".TON(IN := "Etapas_Grafcet".ETAPA_3 OR "Etapas_Grafcet".ETAPA_6 OR "Etapas_Grafcet".ETAPA_9 OR "Etapas_Grafcet".ETAPA_15,
                   PT := "Inputs_HMI".T_POS_EVS);
END_REGION

REGION Network 19: Tempo de lavagem
   RUNG wire#powerrail
      Contact( "Etapas_Grafcet".ETAPA_4 )
      { S7_Templates := "time_type := Time" } "T_LAVAGEM".TONR(r := "Etapas_Grafcet".ETAPA_5, pt := "Inputs_HMI".T_LAVAGEM, et =>)
   END_RUNG
   // the same network as SCL:
   "T_LAVAGEM".TONR(IN := "Etapas_Grafcet".ETAPA_4, R := "Etapas_Grafcet".ETAPA_5, PT := "Inputs_HMI".T_LAVAGEM);
END_REGION

REGION Network 20: Tempo de rinse
   RUNG wire#powerrail
      Contact( "Etapas_Grafcet".ETAPA_7 )
      { S7_Templates := "time_type := Time" } "T_RINSE".TONR(r := "Etapas_Grafcet".ETAPA_8, pt := "Inputs_HMI".T_RINSE, et =>)
   END_RUNG
   // the same network as SCL:
   "T_RINSE".TONR(IN := "Etapas_Grafcet".ETAPA_7, R := "Etapas_Grafcet".ETAPA_8, PT := "Inputs_HMI".T_RINSE);
END_REGION
END_FUNCTION

FUNCTION "Controlo_Ciclo_Limpeza" : Void   // FC2, LAD
{ S7_Optimized_Access := 'TRUE' }
VERSION : 0.1
// stored: AutoNumber true, IsIECCheckEnabled false, SetENOAutomatically false, UDAEnableTagReadback false
   VAR_TEMP   // added for the SCL form of the ladder/FBD networks
      _w1 : Bool;
   END_VAR
BEGIN

REGION Network 1: Hold Etapa 1
   // Devido à etapa 1 fazer reset a si mesma, foi necessário criar esta memória para indicar que tal filtro está em ciclo
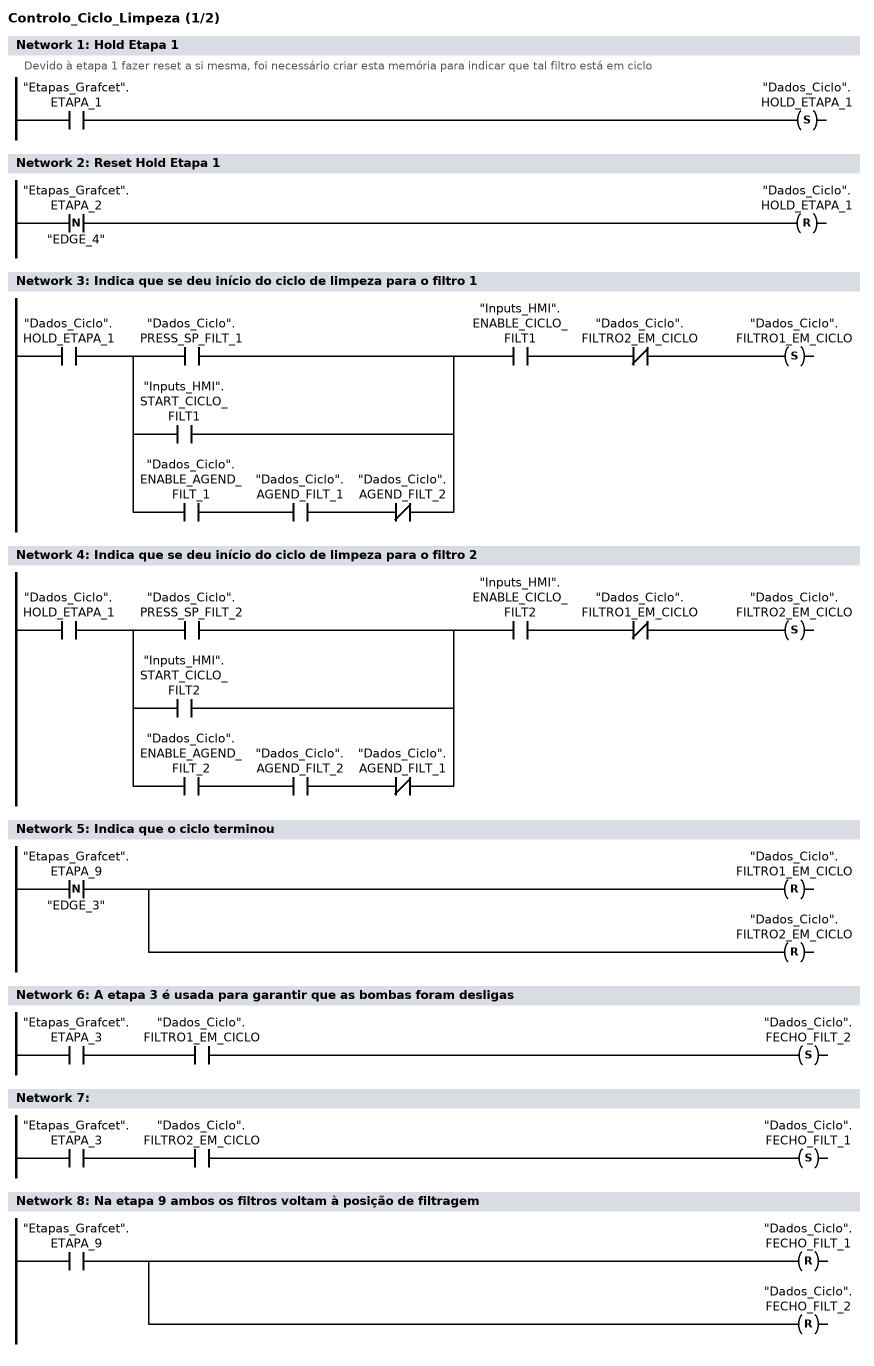
   RUNG wire#powerrail
      Contact( "Etapas_Grafcet".ETAPA_1 )
      S_Coil( "Dados_Ciclo".HOLD_ETAPA_1 )
   END_RUNG
   // the same network as SCL:
   IF "Etapas_Grafcet".ETAPA_1 THEN "Dados_Ciclo".HOLD_ETAPA_1 := TRUE; END_IF;
END_REGION

REGION Network 2: Reset Hold Etapa 1
   RUNG wire#powerrail
      N_Contact(operand := "Etapas_Grafcet".ETAPA_2, bit := "EDGE_4")
      R_Coil( "Dados_Ciclo".HOLD_ETAPA_1 )
   END_RUNG
   // the same network as SCL:
   #_w1 := NOT "Etapas_Grafcet".ETAPA_2 AND "EDGE_4";   // falling edge of "Etapas_Grafcet".ETAPA_2
   "EDGE_4" := "Etapas_Grafcet".ETAPA_2;
   IF #_w1 THEN "Dados_Ciclo".HOLD_ETAPA_1 := FALSE; END_IF;
END_REGION

REGION Network 3: Indica que se deu início do ciclo de limpeza para o filtro 1
   RUNG wire#powerrail
      Contact( "Dados_Ciclo".HOLD_ETAPA_1 )
      wire#w1
      Contact( "Dados_Ciclo".PRESS_SP_FILT_1 )
      wire#w2
      Contact( "Inputs_HMI".ENABLE_CICLO_FILT1 )
      I_Contact( "Dados_Ciclo".FILTRO2_EM_CICLO )
      S_Coil( "Dados_Ciclo".FILTRO1_EM_CICLO )
   END_RUNG
   RUNG wire#w1
      Contact( "Inputs_HMI".START_CICLO_FILT1 )
   END_RUNG wire#w2
   RUNG wire#w1
      Contact( "Dados_Ciclo".ENABLE_AGEND_FILT_1 )
      Contact( "Dados_Ciclo".AGEND_FILT_1 )
      I_Contact( "Dados_Ciclo".AGEND_FILT_2 )
   END_RUNG wire#w2
   // the same network as SCL:
   IF "Dados_Ciclo".HOLD_ETAPA_1 AND ("Dados_Ciclo".PRESS_SP_FILT_1 OR "Inputs_HMI".START_CICLO_FILT1 OR ("Dados_Ciclo".ENABLE_AGEND_FILT_1 AND "Dados_Ciclo".AGEND_FILT_1 AND NOT "Dados_Ciclo".AGEND_FILT_2)) AND "Inputs_HMI".ENABLE_CICLO_FILT1 AND NOT "Dados_Ciclo".FILTRO2_EM_CICLO THEN
       "Dados_Ciclo".FILTRO1_EM_CICLO := TRUE;
   END_IF;
END_REGION

REGION Network 4: Indica que se deu início do ciclo de limpeza para o filtro 2
   RUNG wire#powerrail
      Contact( "Dados_Ciclo".HOLD_ETAPA_1 )
      wire#w1
      Contact( "Dados_Ciclo".PRESS_SP_FILT_2 )
      wire#w2
      Contact( "Inputs_HMI".ENABLE_CICLO_FILT2 )
      I_Contact( "Dados_Ciclo".FILTRO1_EM_CICLO )
      S_Coil( "Dados_Ciclo".FILTRO2_EM_CICLO )
   END_RUNG
   RUNG wire#w1
      Contact( "Inputs_HMI".START_CICLO_FILT2 )
   END_RUNG wire#w2
   RUNG wire#w1
      Contact( "Dados_Ciclo".ENABLE_AGEND_FILT_2 )
      Contact( "Dados_Ciclo".AGEND_FILT_2 )
      I_Contact( "Dados_Ciclo".AGEND_FILT_1 )
   END_RUNG wire#w2
   // the same network as SCL:
   IF "Dados_Ciclo".HOLD_ETAPA_1 AND ("Dados_Ciclo".PRESS_SP_FILT_2 OR "Inputs_HMI".START_CICLO_FILT2 OR ("Dados_Ciclo".ENABLE_AGEND_FILT_2 AND "Dados_Ciclo".AGEND_FILT_2 AND NOT "Dados_Ciclo".AGEND_FILT_1)) AND "Inputs_HMI".ENABLE_CICLO_FILT2 AND NOT "Dados_Ciclo".FILTRO1_EM_CICLO THEN
       "Dados_Ciclo".FILTRO2_EM_CICLO := TRUE;
   END_IF;
END_REGION

REGION Network 5: Indica que o ciclo terminou
   RUNG wire#powerrail
      N_Contact(operand := "Etapas_Grafcet".ETAPA_9, bit := "EDGE_3")
      wire#w1
      R_Coil( "Dados_Ciclo".FILTRO1_EM_CICLO )
   END_RUNG
   RUNG wire#w1
      R_Coil( "Dados_Ciclo".FILTRO2_EM_CICLO )
   END_RUNG
   // the same network as SCL:
   #_w1 := NOT "Etapas_Grafcet".ETAPA_9 AND "EDGE_3";   // falling edge of "Etapas_Grafcet".ETAPA_9
   "EDGE_3" := "Etapas_Grafcet".ETAPA_9;
   IF #_w1 THEN
       "Dados_Ciclo".FILTRO1_EM_CICLO := FALSE;
       "Dados_Ciclo".FILTRO2_EM_CICLO := FALSE;
   END_IF;
END_REGION

REGION Network 6: A etapa 3 é usada para garantir que as bombas foram desligas
   RUNG wire#powerrail
      Contact( "Etapas_Grafcet".ETAPA_3 )
      Contact( "Dados_Ciclo".FILTRO1_EM_CICLO )
      S_Coil( "Dados_Ciclo".FECHO_FILT_2 )
   END_RUNG
   // the same network as SCL:
   IF "Etapas_Grafcet".ETAPA_3 AND "Dados_Ciclo".FILTRO1_EM_CICLO THEN
       "Dados_Ciclo".FECHO_FILT_2 := TRUE;
   END_IF;
END_REGION

REGION Network 7
   RUNG wire#powerrail
      Contact( "Etapas_Grafcet".ETAPA_3 )
      Contact( "Dados_Ciclo".FILTRO2_EM_CICLO )
      S_Coil( "Dados_Ciclo".FECHO_FILT_1 )
   END_RUNG
   // the same network as SCL:
   IF "Etapas_Grafcet".ETAPA_3 AND "Dados_Ciclo".FILTRO2_EM_CICLO THEN
       "Dados_Ciclo".FECHO_FILT_1 := TRUE;
   END_IF;
END_REGION

REGION Network 8: Na etapa 9 ambos os filtros voltam à posição de filtragem
   RUNG wire#powerrail
      Contact( "Etapas_Grafcet".ETAPA_9 )
      wire#w1
      R_Coil( "Dados_Ciclo".FECHO_FILT_1 )
   END_RUNG
   RUNG wire#w1
      R_Coil( "Dados_Ciclo".FECHO_FILT_2 )
   END_RUNG
   // the same network as SCL:
   IF "Etapas_Grafcet".ETAPA_9 THEN
       "Dados_Ciclo".FECHO_FILT_1 := FALSE;
       "Dados_Ciclo".FECHO_FILT_2 := FALSE;
   END_IF;
END_REGION

REGION Network 9: Set à paragem de ciclo
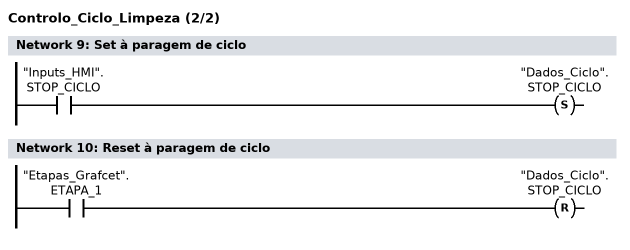
   RUNG wire#powerrail
      Contact( "Inputs_HMI".STOP_CICLO )
      S_Coil( "Dados_Ciclo".STOP_CICLO )
   END_RUNG
   // the same network as SCL:
   IF "Inputs_HMI".STOP_CICLO THEN "Dados_Ciclo".STOP_CICLO := TRUE; END_IF;
END_REGION

REGION Network 10: Reset à paragem de ciclo
   RUNG wire#powerrail
      Contact( "Etapas_Grafcet".ETAPA_1 )
      R_Coil( "Dados_Ciclo".STOP_CICLO )
   END_RUNG
   // the same network as SCL:
   IF "Etapas_Grafcet".ETAPA_1 THEN "Dados_Ciclo".STOP_CICLO := FALSE; END_IF;
END_REGION
END_FUNCTION

FUNCTION "Controlo_Ciclo_Manual" : Void
{ S7_Optimized_Access := 'TRUE' }
VERSION : 0.1

BEGIN
	REGION controlo_etapa_anterior
	    //este bloco serve para saber qual a posição das válvulas antes da passagem para modo manual
	    IF "Etapas_Grafcet".ETAPA_1 = TRUE THEN
	        "Dados_Ciclo".ETAPA_ANTERIOR := 1;
	    END_IF;
	    
	    IF "Etapas_Grafcet".ETAPA_2 = TRUE THEN
	        "Dados_Ciclo".ETAPA_ANTERIOR := 2;
	    END_IF;
	    
	    IF "Etapas_Grafcet".ETAPA_3 = TRUE THEN
	        "Dados_Ciclo".ETAPA_ANTERIOR := 3;
	    END_IF;
	    
	    IF "Etapas_Grafcet".ETAPA_4 = TRUE THEN
	        "Dados_Ciclo".ETAPA_ANTERIOR := 4;
	    END_IF;
	    
	    IF "Etapas_Grafcet".ETAPA_5 = TRUE THEN
	        "Dados_Ciclo".ETAPA_ANTERIOR := 5;
	    END_IF;
	    
	    IF "Etapas_Grafcet".ETAPA_6 = TRUE THEN
	        "Dados_Ciclo".ETAPA_ANTERIOR := 6;
	    END_IF;
	    
	    IF "Etapas_Grafcet".ETAPA_7 = TRUE THEN
	        "Dados_Ciclo".ETAPA_ANTERIOR := 7;
	    END_IF;
	    
	    IF "Etapas_Grafcet".ETAPA_8 = TRUE THEN
	        "Dados_Ciclo".ETAPA_ANTERIOR := 8;
	    END_IF;
	    
	    IF "Etapas_Grafcet".ETAPA_9 = TRUE THEN
	        "Dados_Ciclo".ETAPA_ANTERIOR := 9;
	    END_IF;
	    
	END_REGION
	REGION controlo_etapa_13
	    // este bloco serve para reduzir o numero de contactos na nw13 do ciclo de limpeza
	    IF "Etapas_Grafcet".ETAPA_1 = TRUE OR
	       "Etapas_Grafcet".ETAPA_2 = TRUE OR
	       "Etapas_Grafcet".ETAPA_3 = TRUE OR
	       "Etapas_Grafcet".ETAPA_4 = TRUE OR
	       "Etapas_Grafcet".ETAPA_5 = TRUE OR
	       "Etapas_Grafcet".ETAPA_6 = TRUE OR
	       "Etapas_Grafcet".ETAPA_7 = TRUE OR
	       "Etapas_Grafcet".ETAPA_8 = TRUE OR
	       "Etapas_Grafcet".ETAPA_9 = TRUE
	    THEN
	        "Dados_Ciclo".ETAPA_N := TRUE;
	    END_IF;
	    
	    //reset às etaps de 1 a 9 pela etapa 13
	    IF "Etapas_Grafcet".ETAPA_13 = TRUE
	    THEN
	        "Etapas_Grafcet".ETAPA_1 := FALSE;
	        "Etapas_Grafcet".ETAPA_2 := FALSE;
	        "Etapas_Grafcet".ETAPA_3 := FALSE;
	        "Etapas_Grafcet".ETAPA_4 := FALSE;
	        "Etapas_Grafcet".ETAPA_5 := FALSE;
	        "Etapas_Grafcet".ETAPA_6 := FALSE;
	        "Etapas_Grafcet".ETAPA_7 := FALSE;
	        "Etapas_Grafcet".ETAPA_8 := FALSE;
	        "Etapas_Grafcet".ETAPA_9 := FALSE;
	        
	        "Dados_Ciclo".ETAPA_N := FALSE;
	    END_IF;
	    
	END_REGION
END_FUNCTION

FUNCTION "Saídas_Bombas" : Void   // FC3, LAD
{ S7_Optimized_Access := 'TRUE' }
VERSION : 0.1
// stored: AutoNumber true, IsIECCheckEnabled false, SetENOAutomatically false, UDAEnableTagReadback false
   VAR_TEMP
      BOMBA_1_VAR : Bool;
      BOMBA_2_VAR : Bool;
      BOMBA_3_RESERVA : Bool;
   END_VAR
BEGIN

REGION Network 1: Bomba 1 (com variador)
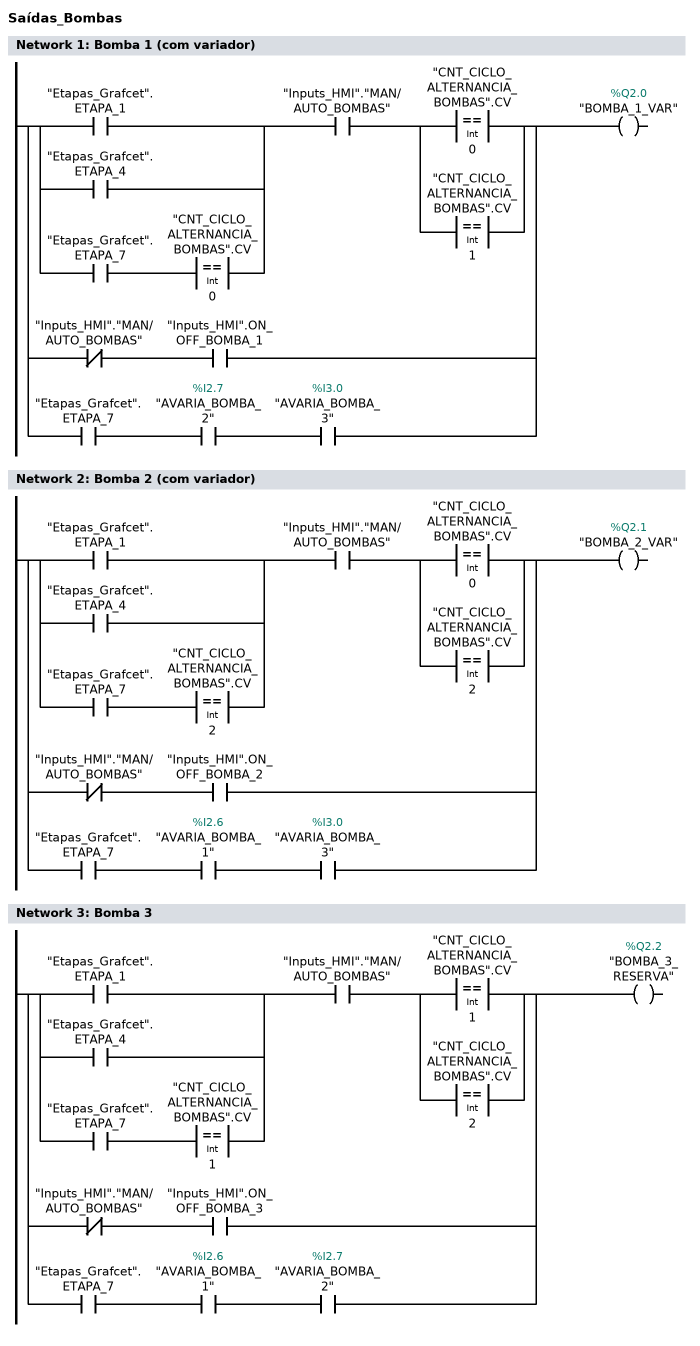
   RUNG wire#powerrail
      Contact( "Etapas_Grafcet".ETAPA_1 )
      wire#w1
      Contact( "Inputs_HMI"."MAN/AUTO_BOMBAS" )
      wire#w2
      { S7_Templates := "SrcType := Int" } EQ_Contact(in1 := "CNT_CICLO_ALTERNANCIA_BOMBAS".CV, in2 := 0)
      wire#w3
      Coil( "BOMBA_1_VAR" )
   END_RUNG
   RUNG wire#powerrail
      Contact( "Etapas_Grafcet".ETAPA_4 )
   END_RUNG wire#w1
   RUNG wire#powerrail
      Contact( "Etapas_Grafcet".ETAPA_7 )
      { S7_Templates := "SrcType := Int" } EQ_Contact(in1 := "CNT_CICLO_ALTERNANCIA_BOMBAS".CV, in2 := 0)
   END_RUNG wire#w1
   RUNG wire#w2
      { S7_Templates := "SrcType := Int" } EQ_Contact(in1 := "CNT_CICLO_ALTERNANCIA_BOMBAS".CV, in2 := 1)
   END_RUNG wire#w3
   RUNG wire#powerrail
      I_Contact( "Inputs_HMI"."MAN/AUTO_BOMBAS" )
      Contact( "Inputs_HMI".ON_OFF_BOMBA_1 )
   END_RUNG wire#w3
   RUNG wire#powerrail
      Contact( "Etapas_Grafcet".ETAPA_7 )
      Contact( "AVARIA_BOMBA_2" )
      Contact( "AVARIA_BOMBA_3" )
   END_RUNG wire#w3
   // the same network as SCL:
   "BOMBA_1_VAR" := (("Etapas_Grafcet".ETAPA_1 OR "Etapas_Grafcet".ETAPA_4 OR ("Etapas_Grafcet".ETAPA_7 AND ("CNT_CICLO_ALTERNANCIA_BOMBAS".CV = 0))) AND "Inputs_HMI"."MAN/AUTO_BOMBAS" AND (("CNT_CICLO_ALTERNANCIA_BOMBAS".CV = 0) OR ("CNT_CICLO_ALTERNANCIA_BOMBAS".CV = 1))) OR (NOT "Inputs_HMI"."MAN/AUTO_BOMBAS" AND "Inputs_HMI".ON_OFF_BOMBA_1) OR ("Etapas_Grafcet".ETAPA_7 AND "AVARIA_BOMBA_2" AND "AVARIA_BOMBA_3");
END_REGION

REGION Network 2: Bomba 2 (com variador)
   RUNG wire#powerrail
      Contact( "Etapas_Grafcet".ETAPA_1 )
      wire#w1
      Contact( "Inputs_HMI"."MAN/AUTO_BOMBAS" )
      wire#w2
      { S7_Templates := "SrcType := Int" } EQ_Contact(in1 := "CNT_CICLO_ALTERNANCIA_BOMBAS".CV, in2 := 0)
      wire#w3
      Coil( "BOMBA_2_VAR" )
   END_RUNG
   RUNG wire#powerrail
      Contact( "Etapas_Grafcet".ETAPA_4 )
   END_RUNG wire#w1
   RUNG wire#powerrail
      Contact( "Etapas_Grafcet".ETAPA_7 )
      { S7_Templates := "SrcType := Int" } EQ_Contact(in1 := "CNT_CICLO_ALTERNANCIA_BOMBAS".CV, in2 := 2)
   END_RUNG wire#w1
   RUNG wire#w2
      { S7_Templates := "SrcType := Int" } EQ_Contact(in1 := "CNT_CICLO_ALTERNANCIA_BOMBAS".CV, in2 := 2)
   END_RUNG wire#w3
   RUNG wire#powerrail
      I_Contact( "Inputs_HMI"."MAN/AUTO_BOMBAS" )
      Contact( "Inputs_HMI".ON_OFF_BOMBA_2 )
   END_RUNG wire#w3
   RUNG wire#powerrail
      Contact( "Etapas_Grafcet".ETAPA_7 )
      Contact( "AVARIA_BOMBA_1" )
      Contact( "AVARIA_BOMBA_3" )
   END_RUNG wire#w3
   // the same network as SCL:
   "BOMBA_2_VAR" := (("Etapas_Grafcet".ETAPA_1 OR "Etapas_Grafcet".ETAPA_4 OR ("Etapas_Grafcet".ETAPA_7 AND ("CNT_CICLO_ALTERNANCIA_BOMBAS".CV = 2))) AND "Inputs_HMI"."MAN/AUTO_BOMBAS" AND (("CNT_CICLO_ALTERNANCIA_BOMBAS".CV = 0) OR ("CNT_CICLO_ALTERNANCIA_BOMBAS".CV = 2))) OR (NOT "Inputs_HMI"."MAN/AUTO_BOMBAS" AND "Inputs_HMI".ON_OFF_BOMBA_2) OR ("Etapas_Grafcet".ETAPA_7 AND "AVARIA_BOMBA_1" AND "AVARIA_BOMBA_3");
END_REGION

REGION Network 3: Bomba 3
   RUNG wire#powerrail
      Contact( "Etapas_Grafcet".ETAPA_1 )
      wire#w1
      Contact( "Inputs_HMI"."MAN/AUTO_BOMBAS" )
      wire#w2
      { S7_Templates := "SrcType := Int" } EQ_Contact(in1 := "CNT_CICLO_ALTERNANCIA_BOMBAS".CV, in2 := 1)
      wire#w3
      Coil( "BOMBA_3_RESERVA" )
   END_RUNG
   RUNG wire#powerrail
      Contact( "Etapas_Grafcet".ETAPA_4 )
   END_RUNG wire#w1
   RUNG wire#powerrail
      Contact( "Etapas_Grafcet".ETAPA_7 )
      { S7_Templates := "SrcType := Int" } EQ_Contact(in1 := "CNT_CICLO_ALTERNANCIA_BOMBAS".CV, in2 := 1)
   END_RUNG wire#w1
   RUNG wire#w2
      { S7_Templates := "SrcType := Int" } EQ_Contact(in1 := "CNT_CICLO_ALTERNANCIA_BOMBAS".CV, in2 := 2)
   END_RUNG wire#w3
   RUNG wire#powerrail
      I_Contact( "Inputs_HMI"."MAN/AUTO_BOMBAS" )
      Contact( "Inputs_HMI".ON_OFF_BOMBA_3 )
   END_RUNG wire#w3
   RUNG wire#powerrail
      Contact( "Etapas_Grafcet".ETAPA_7 )
      Contact( "AVARIA_BOMBA_1" )
      Contact( "AVARIA_BOMBA_2" )
   END_RUNG wire#w3
   // the same network as SCL:
   "BOMBA_3_RESERVA" := (("Etapas_Grafcet".ETAPA_1 OR "Etapas_Grafcet".ETAPA_4 OR ("Etapas_Grafcet".ETAPA_7 AND ("CNT_CICLO_ALTERNANCIA_BOMBAS".CV = 1))) AND "Inputs_HMI"."MAN/AUTO_BOMBAS" AND (("CNT_CICLO_ALTERNANCIA_BOMBAS".CV = 1) OR ("CNT_CICLO_ALTERNANCIA_BOMBAS".CV = 2))) OR (NOT "Inputs_HMI"."MAN/AUTO_BOMBAS" AND "Inputs_HMI".ON_OFF_BOMBA_3) OR ("Etapas_Grafcet".ETAPA_7 AND "AVARIA_BOMBA_1" AND "AVARIA_BOMBA_2");
END_REGION
END_FUNCTION

FUNCTION "Saídas_Bombas_Temporário" : Void   // FC17, LAD
{ S7_Optimized_Access := 'TRUE' }
VERSION : 0.1
// stored: AutoNumber true, IsIECCheckEnabled false, SetENOAutomatically false, UDAEnableTagReadback false
BEGIN

REGION Network 1
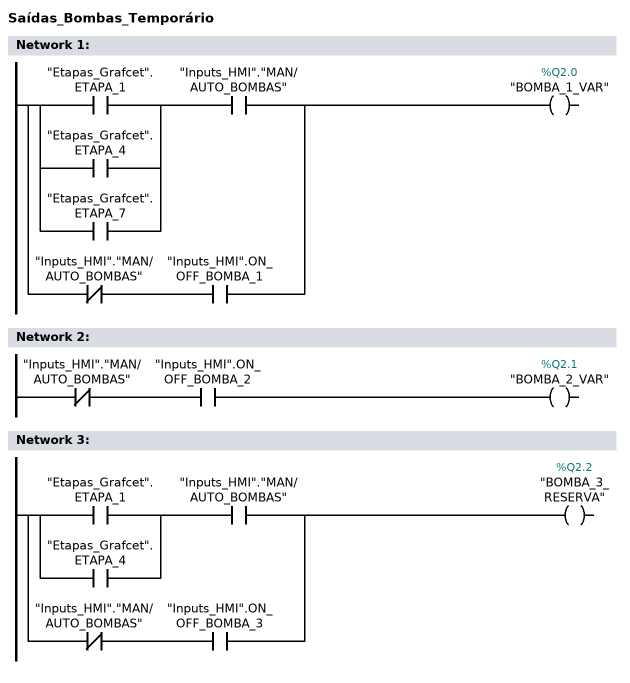
   RUNG wire#powerrail
      Contact( "Etapas_Grafcet".ETAPA_1 )
      wire#w1
      Contact( "Inputs_HMI"."MAN/AUTO_BOMBAS" )
      wire#w2
      Coil( "BOMBA_1_VAR" )
   END_RUNG
   RUNG wire#powerrail
      Contact( "Etapas_Grafcet".ETAPA_4 )
   END_RUNG wire#w1
   RUNG wire#powerrail
      Contact( "Etapas_Grafcet".ETAPA_7 )
   END_RUNG wire#w1
   RUNG wire#powerrail
      I_Contact( "Inputs_HMI"."MAN/AUTO_BOMBAS" )
      Contact( "Inputs_HMI".ON_OFF_BOMBA_1 )
   END_RUNG wire#w2
   // the same network as SCL:
   "BOMBA_1_VAR" := (("Etapas_Grafcet".ETAPA_1 OR "Etapas_Grafcet".ETAPA_4 OR "Etapas_Grafcet".ETAPA_7) AND "Inputs_HMI"."MAN/AUTO_BOMBAS") OR (NOT "Inputs_HMI"."MAN/AUTO_BOMBAS" AND "Inputs_HMI".ON_OFF_BOMBA_1);
END_REGION

REGION Network 2
   RUNG wire#powerrail
      I_Contact( "Inputs_HMI"."MAN/AUTO_BOMBAS" )
      Contact( "Inputs_HMI".ON_OFF_BOMBA_2 )
      Coil( "BOMBA_2_VAR" )
   END_RUNG
   // the same network as SCL:
   "BOMBA_2_VAR" := NOT "Inputs_HMI"."MAN/AUTO_BOMBAS" AND "Inputs_HMI".ON_OFF_BOMBA_2;
END_REGION

REGION Network 3
   RUNG wire#powerrail
      Contact( "Etapas_Grafcet".ETAPA_1 )
      wire#w1
      Contact( "Inputs_HMI"."MAN/AUTO_BOMBAS" )
      wire#w2
      Coil( "BOMBA_3_RESERVA" )
   END_RUNG
   RUNG wire#powerrail
      Contact( "Etapas_Grafcet".ETAPA_4 )
   END_RUNG wire#w1
   RUNG wire#powerrail
      I_Contact( "Inputs_HMI"."MAN/AUTO_BOMBAS" )
      Contact( "Inputs_HMI".ON_OFF_BOMBA_3 )
   END_RUNG wire#w2
   // the same network as SCL:
   "BOMBA_3_RESERVA" := (("Etapas_Grafcet".ETAPA_1 OR "Etapas_Grafcet".ETAPA_4) AND "Inputs_HMI"."MAN/AUTO_BOMBAS") OR (NOT "Inputs_HMI"."MAN/AUTO_BOMBAS" AND "Inputs_HMI".ON_OFF_BOMBA_3);
END_REGION
END_FUNCTION

FUNCTION "Saídas_EV_Filt1" : Void   // FC4, LAD
{ S7_Optimized_Access := 'TRUE' }
VERSION : 0.1
// stored: AutoNumber true, IsIECCheckEnabled false, SetENOAutomatically false, UDAEnableTagReadback false
BEGIN

REGION Network 1
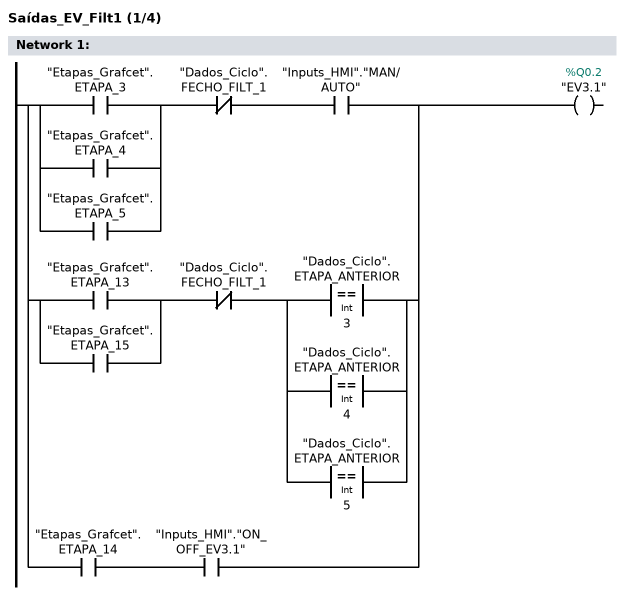
   RUNG wire#powerrail
      Contact( "Etapas_Grafcet".ETAPA_3 )
      wire#w1
      I_Contact( "Dados_Ciclo".FECHO_FILT_1 )
      Contact( "Inputs_HMI"."MAN/AUTO" )
      wire#w2
      Coil( "EV3.1" )
   END_RUNG
   RUNG wire#powerrail
      Contact( "Etapas_Grafcet".ETAPA_4 )
   END_RUNG wire#w1
   RUNG wire#powerrail
      Contact( "Etapas_Grafcet".ETAPA_5 )
   END_RUNG wire#w1
   RUNG wire#powerrail
      Contact( "Etapas_Grafcet".ETAPA_13 )
      wire#w3
      I_Contact( "Dados_Ciclo".FECHO_FILT_1 )
      wire#w4
      { S7_Templates := "SrcType := Int" } EQ_Contact(in1 := "Dados_Ciclo".ETAPA_ANTERIOR, in2 := 3)
   END_RUNG wire#w2
   RUNG wire#powerrail
      Contact( "Etapas_Grafcet".ETAPA_15 )
   END_RUNG wire#w3
   RUNG wire#w4
      { S7_Templates := "SrcType := Int" } EQ_Contact(in1 := "Dados_Ciclo".ETAPA_ANTERIOR, in2 := 4)
   END_RUNG wire#w2
   RUNG wire#w4
      { S7_Templates := "SrcType := Int" } EQ_Contact(in1 := "Dados_Ciclo".ETAPA_ANTERIOR, in2 := 5)
   END_RUNG wire#w2
   RUNG wire#powerrail
      Contact( "Etapas_Grafcet".ETAPA_14 )
      Contact( "Inputs_HMI"."ON_OFF_EV3.1" )
   END_RUNG wire#w2
   // the same network as SCL:
   "EV3.1" := (("Etapas_Grafcet".ETAPA_3 OR "Etapas_Grafcet".ETAPA_4 OR "Etapas_Grafcet".ETAPA_5) AND NOT "Dados_Ciclo".FECHO_FILT_1 AND "Inputs_HMI"."MAN/AUTO") OR (("Etapas_Grafcet".ETAPA_13 OR "Etapas_Grafcet".ETAPA_15) AND NOT "Dados_Ciclo".FECHO_FILT_1 AND (("Dados_Ciclo".ETAPA_ANTERIOR = 3) OR ("Dados_Ciclo".ETAPA_ANTERIOR = 4) OR ("Dados_Ciclo".ETAPA_ANTERIOR = 5))) OR ("Etapas_Grafcet".ETAPA_14 AND "Inputs_HMI"."ON_OFF_EV3.1");
END_REGION

REGION Network 2
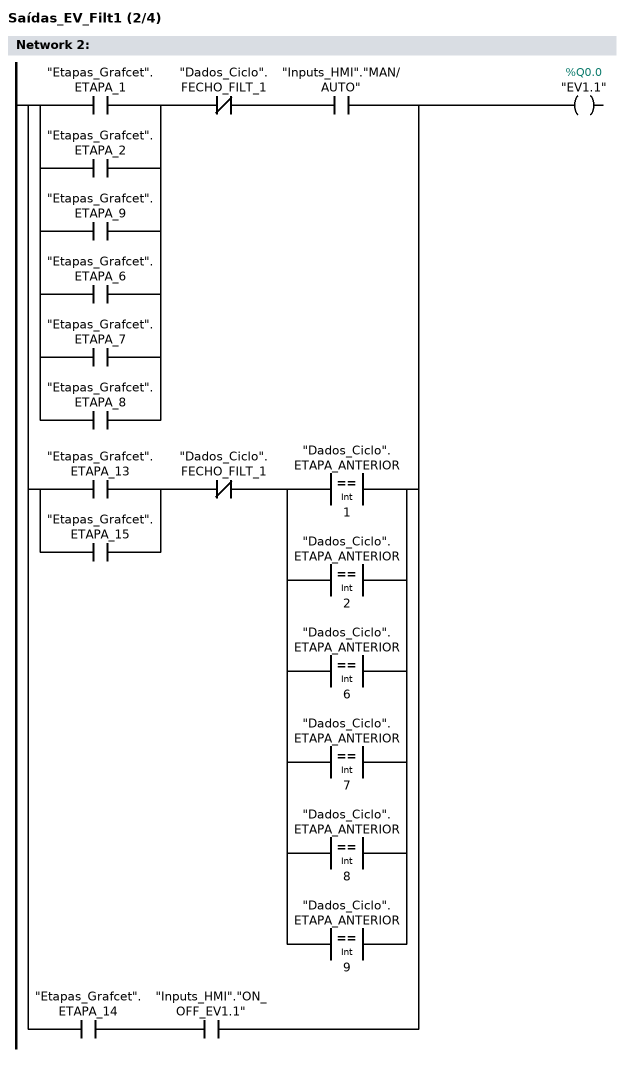
   RUNG wire#powerrail
      Contact( "Etapas_Grafcet".ETAPA_1 )
      wire#w1
      I_Contact( "Dados_Ciclo".FECHO_FILT_1 )
      Contact( "Inputs_HMI"."MAN/AUTO" )
      wire#w2
      Coil( "EV1.1" )
   END_RUNG
   RUNG wire#powerrail
      Contact( "Etapas_Grafcet".ETAPA_2 )
   END_RUNG wire#w1
   RUNG wire#powerrail
      Contact( "Etapas_Grafcet".ETAPA_9 )
   END_RUNG wire#w1
   RUNG wire#powerrail
      Contact( "Etapas_Grafcet".ETAPA_6 )
   END_RUNG wire#w1
   RUNG wire#powerrail
      Contact( "Etapas_Grafcet".ETAPA_7 )
   END_RUNG wire#w1
   RUNG wire#powerrail
      Contact( "Etapas_Grafcet".ETAPA_8 )
   END_RUNG wire#w1
   RUNG wire#powerrail
      Contact( "Etapas_Grafcet".ETAPA_13 )
      wire#w3
      I_Contact( "Dados_Ciclo".FECHO_FILT_1 )
      wire#w4
      { S7_Templates := "SrcType := Int" } EQ_Contact(in1 := "Dados_Ciclo".ETAPA_ANTERIOR, in2 := 1)
   END_RUNG wire#w2
   RUNG wire#powerrail
      Contact( "Etapas_Grafcet".ETAPA_15 )
   END_RUNG wire#w3
   RUNG wire#w4
      { S7_Templates := "SrcType := Int" } EQ_Contact(in1 := "Dados_Ciclo".ETAPA_ANTERIOR, in2 := 2)
   END_RUNG wire#w2
   RUNG wire#w4
      { S7_Templates := "SrcType := Int" } EQ_Contact(in1 := "Dados_Ciclo".ETAPA_ANTERIOR, in2 := 6)
   END_RUNG wire#w2
   RUNG wire#w4
      { S7_Templates := "SrcType := Int" } EQ_Contact(in1 := "Dados_Ciclo".ETAPA_ANTERIOR, in2 := 7)
   END_RUNG wire#w2
   RUNG wire#w4
      { S7_Templates := "SrcType := Int" } EQ_Contact(in1 := "Dados_Ciclo".ETAPA_ANTERIOR, in2 := 8)
   END_RUNG wire#w2
   RUNG wire#w4
      { S7_Templates := "SrcType := Int" } EQ_Contact(in1 := "Dados_Ciclo".ETAPA_ANTERIOR, in2 := 9)
   END_RUNG wire#w2
   RUNG wire#powerrail
      Contact( "Etapas_Grafcet".ETAPA_14 )
      Contact( "Inputs_HMI"."ON_OFF_EV1.1" )
   END_RUNG wire#w2
   // the same network as SCL:
   "EV1.1" := (("Etapas_Grafcet".ETAPA_1 OR "Etapas_Grafcet".ETAPA_2 OR "Etapas_Grafcet".ETAPA_9 OR "Etapas_Grafcet".ETAPA_6 OR "Etapas_Grafcet".ETAPA_7 OR "Etapas_Grafcet".ETAPA_8) AND NOT "Dados_Ciclo".FECHO_FILT_1 AND "Inputs_HMI"."MAN/AUTO") OR (("Etapas_Grafcet".ETAPA_13 OR "Etapas_Grafcet".ETAPA_15) AND NOT "Dados_Ciclo".FECHO_FILT_1 AND (("Dados_Ciclo".ETAPA_ANTERIOR = 1) OR ("Dados_Ciclo".ETAPA_ANTERIOR = 2) OR ("Dados_Ciclo".ETAPA_ANTERIOR = 6) OR ("Dados_Ciclo".ETAPA_ANTERIOR = 7) OR ("Dados_Ciclo".ETAPA_ANTERIOR = 8) OR ("Dados_Ciclo".ETAPA_ANTERIOR = 9))) OR ("Etapas_Grafcet".ETAPA_14 AND "Inputs_HMI"."ON_OFF_EV1.1");
END_REGION

REGION Network 3
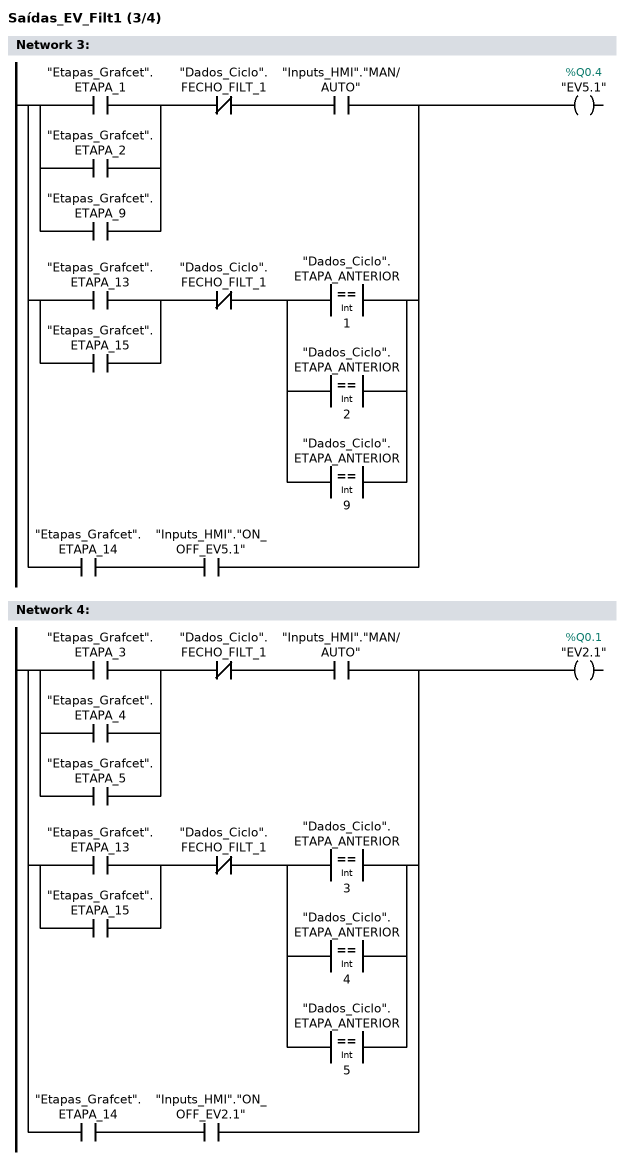
   RUNG wire#powerrail
      Contact( "Etapas_Grafcet".ETAPA_1 )
      wire#w1
      I_Contact( "Dados_Ciclo".FECHO_FILT_1 )
      Contact( "Inputs_HMI"."MAN/AUTO" )
      wire#w2
      Coil( "EV5.1" )
   END_RUNG
   RUNG wire#powerrail
      Contact( "Etapas_Grafcet".ETAPA_2 )
   END_RUNG wire#w1
   RUNG wire#powerrail
      Contact( "Etapas_Grafcet".ETAPA_9 )
   END_RUNG wire#w1
   RUNG wire#powerrail
      Contact( "Etapas_Grafcet".ETAPA_13 )
      wire#w3
      I_Contact( "Dados_Ciclo".FECHO_FILT_1 )
      wire#w4
      { S7_Templates := "SrcType := Int" } EQ_Contact(in1 := "Dados_Ciclo".ETAPA_ANTERIOR, in2 := 1)
   END_RUNG wire#w2
   RUNG wire#powerrail
      Contact( "Etapas_Grafcet".ETAPA_15 )
   END_RUNG wire#w3
   RUNG wire#w4
      { S7_Templates := "SrcType := Int" } EQ_Contact(in1 := "Dados_Ciclo".ETAPA_ANTERIOR, in2 := 2)
   END_RUNG wire#w2
   RUNG wire#w4
      { S7_Templates := "SrcType := Int" } EQ_Contact(in1 := "Dados_Ciclo".ETAPA_ANTERIOR, in2 := 9)
   END_RUNG wire#w2
   RUNG wire#powerrail
      Contact( "Etapas_Grafcet".ETAPA_14 )
      Contact( "Inputs_HMI"."ON_OFF_EV5.1" )
   END_RUNG wire#w2
   // the same network as SCL:
   "EV5.1" := (("Etapas_Grafcet".ETAPA_1 OR "Etapas_Grafcet".ETAPA_2 OR "Etapas_Grafcet".ETAPA_9) AND NOT "Dados_Ciclo".FECHO_FILT_1 AND "Inputs_HMI"."MAN/AUTO") OR (("Etapas_Grafcet".ETAPA_13 OR "Etapas_Grafcet".ETAPA_15) AND NOT "Dados_Ciclo".FECHO_FILT_1 AND (("Dados_Ciclo".ETAPA_ANTERIOR = 1) OR ("Dados_Ciclo".ETAPA_ANTERIOR = 2) OR ("Dados_Ciclo".ETAPA_ANTERIOR = 9))) OR ("Etapas_Grafcet".ETAPA_14 AND "Inputs_HMI"."ON_OFF_EV5.1");
END_REGION

REGION Network 4
   RUNG wire#powerrail
      Contact( "Etapas_Grafcet".ETAPA_3 )
      wire#w1
      I_Contact( "Dados_Ciclo".FECHO_FILT_1 )
      Contact( "Inputs_HMI"."MAN/AUTO" )
      wire#w2
      Coil( "EV2.1" )
   END_RUNG
   RUNG wire#powerrail
      Contact( "Etapas_Grafcet".ETAPA_4 )
   END_RUNG wire#w1
   RUNG wire#powerrail
      Contact( "Etapas_Grafcet".ETAPA_5 )
   END_RUNG wire#w1
   RUNG wire#powerrail
      Contact( "Etapas_Grafcet".ETAPA_13 )
      wire#w3
      I_Contact( "Dados_Ciclo".FECHO_FILT_1 )
      wire#w4
      { S7_Templates := "SrcType := Int" } EQ_Contact(in1 := "Dados_Ciclo".ETAPA_ANTERIOR, in2 := 3)
   END_RUNG wire#w2
   RUNG wire#powerrail
      Contact( "Etapas_Grafcet".ETAPA_15 )
   END_RUNG wire#w3
   RUNG wire#w4
      { S7_Templates := "SrcType := Int" } EQ_Contact(in1 := "Dados_Ciclo".ETAPA_ANTERIOR, in2 := 4)
   END_RUNG wire#w2
   RUNG wire#w4
      { S7_Templates := "SrcType := Int" } EQ_Contact(in1 := "Dados_Ciclo".ETAPA_ANTERIOR, in2 := 5)
   END_RUNG wire#w2
   RUNG wire#powerrail
      Contact( "Etapas_Grafcet".ETAPA_14 )
      Contact( "Inputs_HMI"."ON_OFF_EV2.1" )
   END_RUNG wire#w2
   // the same network as SCL:
   "EV2.1" := (("Etapas_Grafcet".ETAPA_3 OR "Etapas_Grafcet".ETAPA_4 OR "Etapas_Grafcet".ETAPA_5) AND NOT "Dados_Ciclo".FECHO_FILT_1 AND "Inputs_HMI"."MAN/AUTO") OR (("Etapas_Grafcet".ETAPA_13 OR "Etapas_Grafcet".ETAPA_15) AND NOT "Dados_Ciclo".FECHO_FILT_1 AND (("Dados_Ciclo".ETAPA_ANTERIOR = 3) OR ("Dados_Ciclo".ETAPA_ANTERIOR = 4) OR ("Dados_Ciclo".ETAPA_ANTERIOR = 5))) OR ("Etapas_Grafcet".ETAPA_14 AND "Inputs_HMI"."ON_OFF_EV2.1");
END_REGION

REGION Network 5
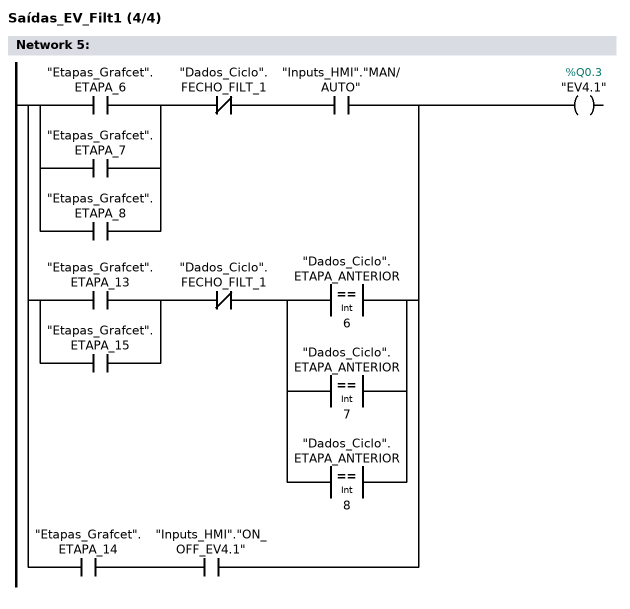
   RUNG wire#powerrail
      Contact( "Etapas_Grafcet".ETAPA_6 )
      wire#w1
      I_Contact( "Dados_Ciclo".FECHO_FILT_1 )
      Contact( "Inputs_HMI"."MAN/AUTO" )
      wire#w2
      Coil( "EV4.1" )
   END_RUNG
   RUNG wire#powerrail
      Contact( "Etapas_Grafcet".ETAPA_7 )
   END_RUNG wire#w1
   RUNG wire#powerrail
      Contact( "Etapas_Grafcet".ETAPA_8 )
   END_RUNG wire#w1
   RUNG wire#powerrail
      Contact( "Etapas_Grafcet".ETAPA_13 )
      wire#w3
      I_Contact( "Dados_Ciclo".FECHO_FILT_1 )
      wire#w4
      { S7_Templates := "SrcType := Int" } EQ_Contact(in1 := "Dados_Ciclo".ETAPA_ANTERIOR, in2 := 6)
   END_RUNG wire#w2
   RUNG wire#powerrail
      Contact( "Etapas_Grafcet".ETAPA_15 )
   END_RUNG wire#w3
   RUNG wire#w4
      { S7_Templates := "SrcType := Int" } EQ_Contact(in1 := "Dados_Ciclo".ETAPA_ANTERIOR, in2 := 7)
   END_RUNG wire#w2
   RUNG wire#w4
      { S7_Templates := "SrcType := Int" } EQ_Contact(in1 := "Dados_Ciclo".ETAPA_ANTERIOR, in2 := 8)
   END_RUNG wire#w2
   RUNG wire#powerrail
      Contact( "Etapas_Grafcet".ETAPA_14 )
      Contact( "Inputs_HMI"."ON_OFF_EV4.1" )
   END_RUNG wire#w2
   // the same network as SCL:
   "EV4.1" := (("Etapas_Grafcet".ETAPA_6 OR "Etapas_Grafcet".ETAPA_7 OR "Etapas_Grafcet".ETAPA_8) AND NOT "Dados_Ciclo".FECHO_FILT_1 AND "Inputs_HMI"."MAN/AUTO") OR (("Etapas_Grafcet".ETAPA_13 OR "Etapas_Grafcet".ETAPA_15) AND NOT "Dados_Ciclo".FECHO_FILT_1 AND (("Dados_Ciclo".ETAPA_ANTERIOR = 6) OR ("Dados_Ciclo".ETAPA_ANTERIOR = 7) OR ("Dados_Ciclo".ETAPA_ANTERIOR = 8))) OR ("Etapas_Grafcet".ETAPA_14 AND "Inputs_HMI"."ON_OFF_EV4.1");
END_REGION
END_FUNCTION

FUNCTION "Saídas_EV_Filt2" : Void   // FC5, LAD
{ S7_Optimized_Access := 'TRUE' }
VERSION : 0.1
// stored: AutoNumber true, IsIECCheckEnabled false, SetENOAutomatically false, UDAEnableTagReadback false
BEGIN

REGION Network 1
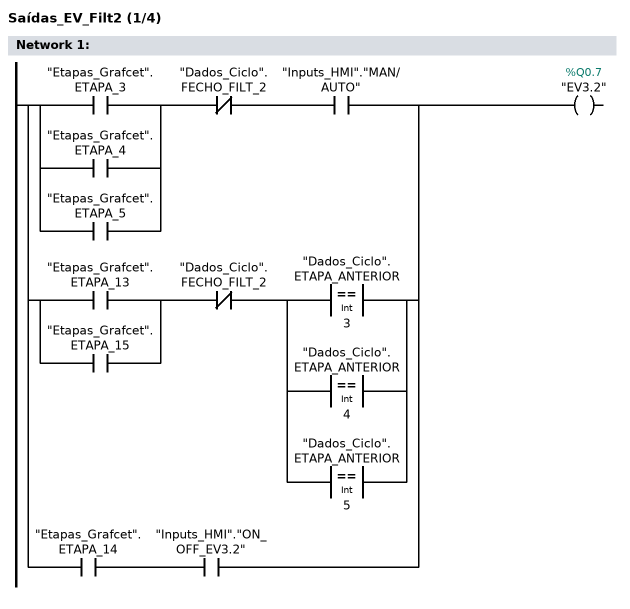
   RUNG wire#powerrail
      Contact( "Etapas_Grafcet".ETAPA_3 )
      wire#w1
      I_Contact( "Dados_Ciclo".FECHO_FILT_2 )
      Contact( "Inputs_HMI"."MAN/AUTO" )
      wire#w2
      Coil( "EV3.2" )
   END_RUNG
   RUNG wire#powerrail
      Contact( "Etapas_Grafcet".ETAPA_4 )
   END_RUNG wire#w1
   RUNG wire#powerrail
      Contact( "Etapas_Grafcet".ETAPA_5 )
   END_RUNG wire#w1
   RUNG wire#powerrail
      Contact( "Etapas_Grafcet".ETAPA_13 )
      wire#w3
      I_Contact( "Dados_Ciclo".FECHO_FILT_2 )
      wire#w4
      { S7_Templates := "SrcType := Int" } EQ_Contact(in1 := "Dados_Ciclo".ETAPA_ANTERIOR, in2 := 3)
   END_RUNG wire#w2
   RUNG wire#powerrail
      Contact( "Etapas_Grafcet".ETAPA_15 )
   END_RUNG wire#w3
   RUNG wire#w4
      { S7_Templates := "SrcType := Int" } EQ_Contact(in1 := "Dados_Ciclo".ETAPA_ANTERIOR, in2 := 4)
   END_RUNG wire#w2
   RUNG wire#w4
      { S7_Templates := "SrcType := Int" } EQ_Contact(in1 := "Dados_Ciclo".ETAPA_ANTERIOR, in2 := 5)
   END_RUNG wire#w2
   RUNG wire#powerrail
      Contact( "Etapas_Grafcet".ETAPA_14 )
      Contact( "Inputs_HMI"."ON_OFF_EV3.2" )
   END_RUNG wire#w2
   // the same network as SCL:
   "EV3.2" := (("Etapas_Grafcet".ETAPA_3 OR "Etapas_Grafcet".ETAPA_4 OR "Etapas_Grafcet".ETAPA_5) AND NOT "Dados_Ciclo".FECHO_FILT_2 AND "Inputs_HMI"."MAN/AUTO") OR (("Etapas_Grafcet".ETAPA_13 OR "Etapas_Grafcet".ETAPA_15) AND NOT "Dados_Ciclo".FECHO_FILT_2 AND (("Dados_Ciclo".ETAPA_ANTERIOR = 3) OR ("Dados_Ciclo".ETAPA_ANTERIOR = 4) OR ("Dados_Ciclo".ETAPA_ANTERIOR = 5))) OR ("Etapas_Grafcet".ETAPA_14 AND "Inputs_HMI"."ON_OFF_EV3.2");
END_REGION

REGION Network 2
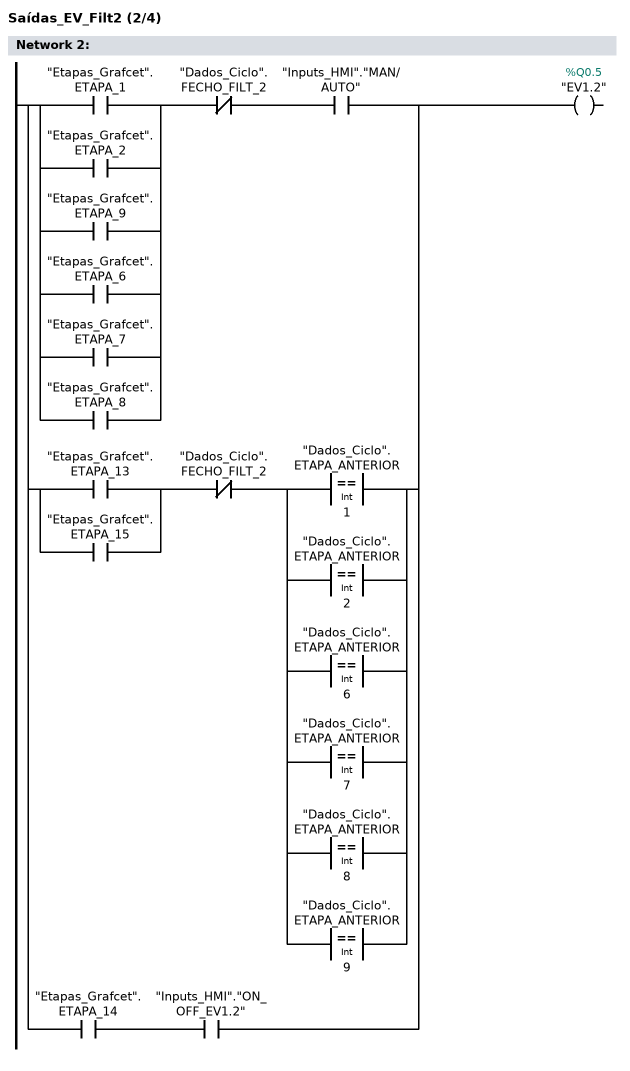
   RUNG wire#powerrail
      Contact( "Etapas_Grafcet".ETAPA_1 )
      wire#w1
      I_Contact( "Dados_Ciclo".FECHO_FILT_2 )
      Contact( "Inputs_HMI"."MAN/AUTO" )
      wire#w2
      Coil( "EV1.2" )
   END_RUNG
   RUNG wire#powerrail
      Contact( "Etapas_Grafcet".ETAPA_2 )
   END_RUNG wire#w1
   RUNG wire#powerrail
      Contact( "Etapas_Grafcet".ETAPA_9 )
   END_RUNG wire#w1
   RUNG wire#powerrail
      Contact( "Etapas_Grafcet".ETAPA_6 )
   END_RUNG wire#w1
   RUNG wire#powerrail
      Contact( "Etapas_Grafcet".ETAPA_7 )
   END_RUNG wire#w1
   RUNG wire#powerrail
      Contact( "Etapas_Grafcet".ETAPA_8 )
   END_RUNG wire#w1
   RUNG wire#powerrail
      Contact( "Etapas_Grafcet".ETAPA_13 )
      wire#w3
      I_Contact( "Dados_Ciclo".FECHO_FILT_2 )
      wire#w4
      { S7_Templates := "SrcType := Int" } EQ_Contact(in1 := "Dados_Ciclo".ETAPA_ANTERIOR, in2 := 1)
   END_RUNG wire#w2
   RUNG wire#powerrail
      Contact( "Etapas_Grafcet".ETAPA_15 )
   END_RUNG wire#w3
   RUNG wire#w4
      { S7_Templates := "SrcType := Int" } EQ_Contact(in1 := "Dados_Ciclo".ETAPA_ANTERIOR, in2 := 2)
   END_RUNG wire#w2
   RUNG wire#w4
      { S7_Templates := "SrcType := Int" } EQ_Contact(in1 := "Dados_Ciclo".ETAPA_ANTERIOR, in2 := 6)
   END_RUNG wire#w2
   RUNG wire#w4
      { S7_Templates := "SrcType := Int" } EQ_Contact(in1 := "Dados_Ciclo".ETAPA_ANTERIOR, in2 := 7)
   END_RUNG wire#w2
   RUNG wire#w4
      { S7_Templates := "SrcType := Int" } EQ_Contact(in1 := "Dados_Ciclo".ETAPA_ANTERIOR, in2 := 8)
   END_RUNG wire#w2
   RUNG wire#w4
      { S7_Templates := "SrcType := Int" } EQ_Contact(in1 := "Dados_Ciclo".ETAPA_ANTERIOR, in2 := 9)
   END_RUNG wire#w2
   RUNG wire#powerrail
      Contact( "Etapas_Grafcet".ETAPA_14 )
      Contact( "Inputs_HMI"."ON_OFF_EV1.2" )
   END_RUNG wire#w2
   // the same network as SCL:
   "EV1.2" := (("Etapas_Grafcet".ETAPA_1 OR "Etapas_Grafcet".ETAPA_2 OR "Etapas_Grafcet".ETAPA_9 OR "Etapas_Grafcet".ETAPA_6 OR "Etapas_Grafcet".ETAPA_7 OR "Etapas_Grafcet".ETAPA_8) AND NOT "Dados_Ciclo".FECHO_FILT_2 AND "Inputs_HMI"."MAN/AUTO") OR (("Etapas_Grafcet".ETAPA_13 OR "Etapas_Grafcet".ETAPA_15) AND NOT "Dados_Ciclo".FECHO_FILT_2 AND (("Dados_Ciclo".ETAPA_ANTERIOR = 1) OR ("Dados_Ciclo".ETAPA_ANTERIOR = 2) OR ("Dados_Ciclo".ETAPA_ANTERIOR = 6) OR ("Dados_Ciclo".ETAPA_ANTERIOR = 7) OR ("Dados_Ciclo".ETAPA_ANTERIOR = 8) OR ("Dados_Ciclo".ETAPA_ANTERIOR = 9))) OR ("Etapas_Grafcet".ETAPA_14 AND "Inputs_HMI"."ON_OFF_EV1.2");
END_REGION

REGION Network 3
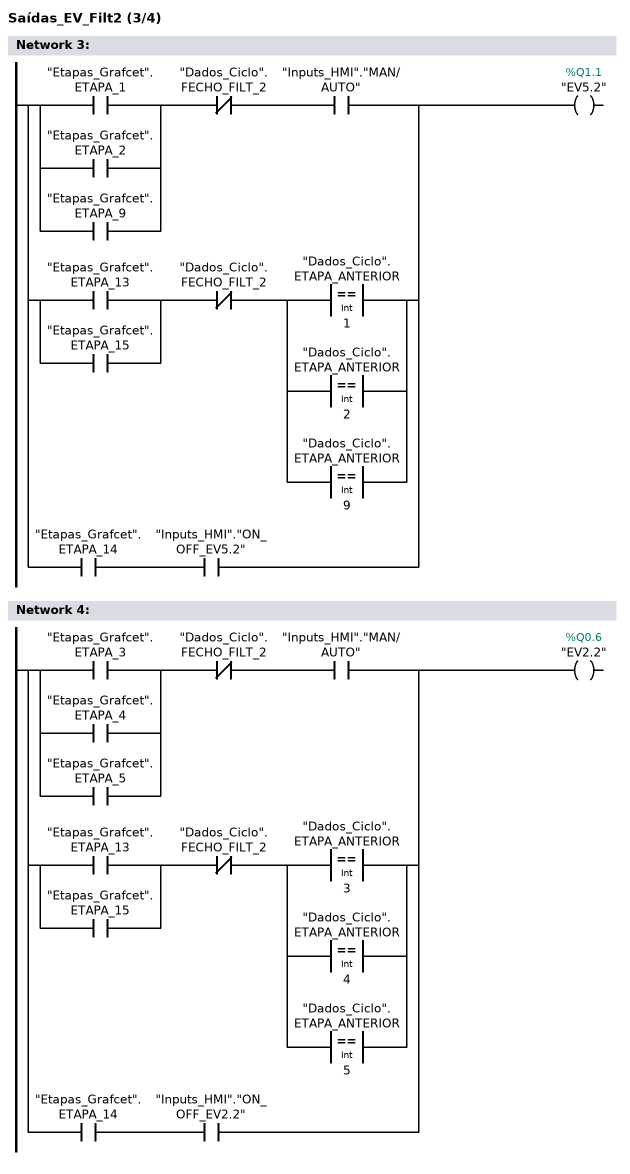
   RUNG wire#powerrail
      Contact( "Etapas_Grafcet".ETAPA_1 )
      wire#w1
      I_Contact( "Dados_Ciclo".FECHO_FILT_2 )
      Contact( "Inputs_HMI"."MAN/AUTO" )
      wire#w2
      Coil( "EV5.2" )
   END_RUNG
   RUNG wire#powerrail
      Contact( "Etapas_Grafcet".ETAPA_2 )
   END_RUNG wire#w1
   RUNG wire#powerrail
      Contact( "Etapas_Grafcet".ETAPA_9 )
   END_RUNG wire#w1
   RUNG wire#powerrail
      Contact( "Etapas_Grafcet".ETAPA_13 )
      wire#w3
      I_Contact( "Dados_Ciclo".FECHO_FILT_2 )
      wire#w4
      { S7_Templates := "SrcType := Int" } EQ_Contact(in1 := "Dados_Ciclo".ETAPA_ANTERIOR, in2 := 1)
   END_RUNG wire#w2
   RUNG wire#powerrail
      Contact( "Etapas_Grafcet".ETAPA_15 )
   END_RUNG wire#w3
   RUNG wire#w4
      { S7_Templates := "SrcType := Int" } EQ_Contact(in1 := "Dados_Ciclo".ETAPA_ANTERIOR, in2 := 2)
   END_RUNG wire#w2
   RUNG wire#w4
      { S7_Templates := "SrcType := Int" } EQ_Contact(in1 := "Dados_Ciclo".ETAPA_ANTERIOR, in2 := 9)
   END_RUNG wire#w2
   RUNG wire#powerrail
      Contact( "Etapas_Grafcet".ETAPA_14 )
      Contact( "Inputs_HMI"."ON_OFF_EV5.2" )
   END_RUNG wire#w2
   // the same network as SCL:
   "EV5.2" := (("Etapas_Grafcet".ETAPA_1 OR "Etapas_Grafcet".ETAPA_2 OR "Etapas_Grafcet".ETAPA_9) AND NOT "Dados_Ciclo".FECHO_FILT_2 AND "Inputs_HMI"."MAN/AUTO") OR (("Etapas_Grafcet".ETAPA_13 OR "Etapas_Grafcet".ETAPA_15) AND NOT "Dados_Ciclo".FECHO_FILT_2 AND (("Dados_Ciclo".ETAPA_ANTERIOR = 1) OR ("Dados_Ciclo".ETAPA_ANTERIOR = 2) OR ("Dados_Ciclo".ETAPA_ANTERIOR = 9))) OR ("Etapas_Grafcet".ETAPA_14 AND "Inputs_HMI"."ON_OFF_EV5.2");
END_REGION

REGION Network 4
   RUNG wire#powerrail
      Contact( "Etapas_Grafcet".ETAPA_3 )
      wire#w1
      I_Contact( "Dados_Ciclo".FECHO_FILT_2 )
      Contact( "Inputs_HMI"."MAN/AUTO" )
      wire#w2
      Coil( "EV2.2" )
   END_RUNG
   RUNG wire#powerrail
      Contact( "Etapas_Grafcet".ETAPA_4 )
   END_RUNG wire#w1
   RUNG wire#powerrail
      Contact( "Etapas_Grafcet".ETAPA_5 )
   END_RUNG wire#w1
   RUNG wire#powerrail
      Contact( "Etapas_Grafcet".ETAPA_13 )
      wire#w3
      I_Contact( "Dados_Ciclo".FECHO_FILT_2 )
      wire#w4
      { S7_Templates := "SrcType := Int" } EQ_Contact(in1 := "Dados_Ciclo".ETAPA_ANTERIOR, in2 := 3)
   END_RUNG wire#w2
   RUNG wire#powerrail
      Contact( "Etapas_Grafcet".ETAPA_15 )
   END_RUNG wire#w3
   RUNG wire#w4
      { S7_Templates := "SrcType := Int" } EQ_Contact(in1 := "Dados_Ciclo".ETAPA_ANTERIOR, in2 := 4)
   END_RUNG wire#w2
   RUNG wire#w4
      { S7_Templates := "SrcType := Int" } EQ_Contact(in1 := "Dados_Ciclo".ETAPA_ANTERIOR, in2 := 5)
   END_RUNG wire#w2
   RUNG wire#powerrail
      Contact( "Etapas_Grafcet".ETAPA_14 )
      Contact( "Inputs_HMI"."ON_OFF_EV2.2" )
   END_RUNG wire#w2
   // the same network as SCL:
   "EV2.2" := (("Etapas_Grafcet".ETAPA_3 OR "Etapas_Grafcet".ETAPA_4 OR "Etapas_Grafcet".ETAPA_5) AND NOT "Dados_Ciclo".FECHO_FILT_2 AND "Inputs_HMI"."MAN/AUTO") OR (("Etapas_Grafcet".ETAPA_13 OR "Etapas_Grafcet".ETAPA_15) AND NOT "Dados_Ciclo".FECHO_FILT_2 AND (("Dados_Ciclo".ETAPA_ANTERIOR = 3) OR ("Dados_Ciclo".ETAPA_ANTERIOR = 4) OR ("Dados_Ciclo".ETAPA_ANTERIOR = 5))) OR ("Etapas_Grafcet".ETAPA_14 AND "Inputs_HMI"."ON_OFF_EV2.2");
END_REGION

REGION Network 5
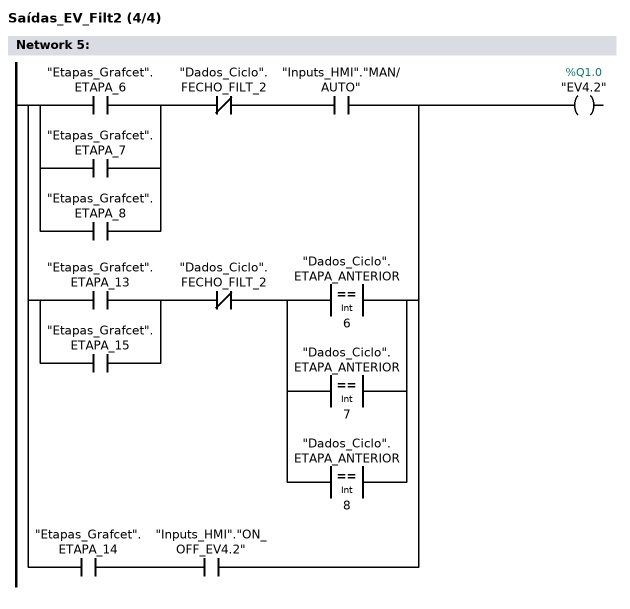
   RUNG wire#powerrail
      Contact( "Etapas_Grafcet".ETAPA_6 )
      wire#w1
      I_Contact( "Dados_Ciclo".FECHO_FILT_2 )
      Contact( "Inputs_HMI"."MAN/AUTO" )
      wire#w2
      Coil( "EV4.2" )
   END_RUNG
   RUNG wire#powerrail
      Contact( "Etapas_Grafcet".ETAPA_7 )
   END_RUNG wire#w1
   RUNG wire#powerrail
      Contact( "Etapas_Grafcet".ETAPA_8 )
   END_RUNG wire#w1
   RUNG wire#powerrail
      Contact( "Etapas_Grafcet".ETAPA_13 )
      wire#w3
      I_Contact( "Dados_Ciclo".FECHO_FILT_2 )
      wire#w4
      { S7_Templates := "SrcType := Int" } EQ_Contact(in1 := "Dados_Ciclo".ETAPA_ANTERIOR, in2 := 6)
   END_RUNG wire#w2
   RUNG wire#powerrail
      Contact( "Etapas_Grafcet".ETAPA_15 )
   END_RUNG wire#w3
   RUNG wire#w4
      { S7_Templates := "SrcType := Int" } EQ_Contact(in1 := "Dados_Ciclo".ETAPA_ANTERIOR, in2 := 7)
   END_RUNG wire#w2
   RUNG wire#w4
      { S7_Templates := "SrcType := Int" } EQ_Contact(in1 := "Dados_Ciclo".ETAPA_ANTERIOR, in2 := 8)
   END_RUNG wire#w2
   RUNG wire#powerrail
      Contact( "Etapas_Grafcet".ETAPA_14 )
      Contact( "Inputs_HMI"."ON_OFF_EV4.2" )
   END_RUNG wire#w2
   // the same network as SCL:
   "EV4.2" := (("Etapas_Grafcet".ETAPA_6 OR "Etapas_Grafcet".ETAPA_7 OR "Etapas_Grafcet".ETAPA_8) AND NOT "Dados_Ciclo".FECHO_FILT_2 AND "Inputs_HMI"."MAN/AUTO") OR (("Etapas_Grafcet".ETAPA_13 OR "Etapas_Grafcet".ETAPA_15) AND NOT "Dados_Ciclo".FECHO_FILT_2 AND (("Dados_Ciclo".ETAPA_ANTERIOR = 6) OR ("Dados_Ciclo".ETAPA_ANTERIOR = 7) OR ("Dados_Ciclo".ETAPA_ANTERIOR = 8))) OR ("Etapas_Grafcet".ETAPA_14 AND "Inputs_HMI"."ON_OFF_EV4.2");
END_REGION
END_FUNCTION

FUNCTION "Posição_EVs" : Void
{ S7_Optimized_Access := 'TRUE' }
VERSION : 0.1
   VAR_TEMP 
      "temp_clock_0.625Hz" : Int;
      "avaria_ev1.1" : Bool;
      "avaria_ev2.1" : Bool;
      "avaria_ev3.1" : Bool;
      "avaria_ev4.1" : Bool;
      "avaria_ev5.1" : Bool;
      "avaria_ev1.2" : Bool;
      "avaria_ev2.2" : Bool;
      "avaria_ev3.2" : Bool;
      "avaria_ev4.2" : Bool;
      "avaria_ev5.2" : Bool;
   END_VAR


BEGIN
	REGION POSICAO_FILTRO_1
	    IF "EV1.1_ABERTA" = TRUE AND "EV5.1_ABERTA" = TRUE AND
	        "EV2.1_FECHADA" = TRUE AND "EV4.1_FECHADA" = TRUE AND
	        "EV3.1_FECHADA" = TRUE AND
	        
	        "EV1.1_FECHADA" = FALSE AND "EV5.1_FECHADA" = FALSE AND
	        "EV2.1_ABERTA" = FALSE AND "EV4.1_ABERTA" = FALSE AND
	        "EV3.1_ABERTA" = FALSE
	    THEN
	        "Dados_Ciclo".POS_EVS_FILT_1 := 'FILTRACAO';
	    ELSE
	        
	        IF "EV2.1_ABERTA" = TRUE AND "EV3.1_ABERTA" = TRUE AND
	            "EV1.1_FECHADA" = TRUE AND "EV4.1_FECHADA" = TRUE AND
	            "EV5.1_FECHADA" = TRUE AND
	            
	            "EV2.1_FECHADA" = FALSE AND "EV3.1_FECHADA" = FALSE AND
	            "EV1.1_ABERTA" = FALSE AND "EV4.1_ABERTA" = FALSE AND
	            "EV5.1_ABERTA" = FALSE
	        THEN
	            "Dados_Ciclo".POS_EVS_FILT_1 := 'LAVAGEM';
	        ELSE
	            
	            IF "EV1.1_ABERTA" = TRUE AND "EV4.1_ABERTA" = TRUE AND
	                "EV2.1_FECHADA" = TRUE AND "EV3.1_FECHADA" = TRUE AND
	                "EV5.1_FECHADA" = TRUE AND
	                
	                "EV1.1_FECHADA" = FALSE AND "EV4.1_FECHADA" = FALSE AND
	                "EV2.1_ABERTA" = FALSE AND "EV3.1_ABERTA" = FALSE AND
	                "EV5.1_ABERTA" = FALSE
	            THEN
	                "Dados_Ciclo".POS_EVS_FILT_1 := 'RINSE';
	            ELSE
	                
	                IF "EV1.1_ABERTA" = TRUE AND "EV3.1_ABERTA" = TRUE AND
	                    "EV2.1_FECHADA" = TRUE AND "EV4.1_FECHADA" = TRUE AND
	                    "EV5.1_FECHADA" = TRUE AND
	                    
	                    "EV1.1_FECHADA" = FALSE AND "EV3.1_FECHADA" = FALSE AND
	                    "EV2.1_ABERTA" = FALSE AND "EV4.1_ABERTA" = FALSE AND
	                    "EV5.1_ABERTA" = FALSE
	                THEN
	                    "Dados_Ciclo".POS_EVS_FILT_1 := 'ESVAZIAMENTO';
	                ELSE
	                    
	                    IF "EV1.1_FECHADA" = TRUE AND "EV2.1_FECHADA" = TRUE AND
	                        "EV3.1_FECHADA" = TRUE AND "EV4.1_FECHADA" = TRUE AND
	                        "EV5.1_FECHADA" = TRUE AND
	                        
	                        "EV1.1_ABERTA" = FALSE AND "EV2.1_ABERTA" = FALSE AND
	                        "EV3.1_ABERTA" = FALSE AND "EV4.1_ABERTA" = FALSE AND
	                        "EV5.1_ABERTA" = FALSE
	                    THEN
	                        "Dados_Ciclo".POS_EVS_FILT_1 := 'FECHO';
	                    ELSE
	                        "Dados_Ciclo".POS_EVS_FILT_1 := 'NULL';
	                    END_IF;
	                END_IF;
	            END_IF;
	        END_IF;
	    END_IF;
	    
	END_REGION
	
	REGION POSICAO_FILTRO_2
	    IF "EV1.2_ABERTA" = TRUE AND "EV5.2_ABERTA" = TRUE AND
	        "EV2.2_FECHADA" = TRUE AND "EV4.2_FECHADA" = TRUE AND
	        "EV3.2_FECHADA" = TRUE AND
	        
	        "EV1.2_FECHADA" = FALSE AND "EV5.2_FECHADA" = FALSE AND
	        "EV2.2_ABERTA" = FALSE AND "EV4.2_ABERTA" = FALSE AND
	        "EV3.2_ABERTA" = FALSE
	    THEN
	        "Dados_Ciclo".POS_EVS_FILT_2 := 'FILTRACAO';
	    ELSE
	        
	        IF "EV2.2_ABERTA" = TRUE AND "EV3.2_ABERTA" = TRUE AND
	            "EV1.2_FECHADA" = TRUE AND "EV4.2_FECHADA" = TRUE AND
	            "EV5.2_FECHADA" = TRUE AND
	            
	            "EV2.2_FECHADA" = FALSE AND "EV3.2_FECHADA" = FALSE AND
	            "EV1.2_ABERTA" = FALSE AND "EV4.2_ABERTA" = FALSE AND
	            "EV5.2_ABERTA" = FALSE
	        THEN
	            "Dados_Ciclo".POS_EVS_FILT_2 := 'LAVAGEM';
	        ELSE
	            
	            IF "EV1.2_ABERTA" = TRUE AND "EV4.2_ABERTA" = TRUE AND
	                "EV2.2_FECHADA" = TRUE AND "EV3.2_FECHADA" = TRUE AND
	                "EV5.2_FECHADA" = TRUE AND
	                
	                "EV1.2_FECHADA" = FALSE AND "EV4.2_FECHADA" = FALSE AND
	                "EV2.2_ABERTA" = FALSE AND "EV3.2_ABERTA" = FALSE AND
	                "EV5.2_ABERTA" = FALSE
	            THEN
	                "Dados_Ciclo".POS_EVS_FILT_2 := 'RINSE';
	            ELSE
	                
	                IF "EV1.2_ABERTA" = TRUE AND "EV3.2_ABERTA" = TRUE AND
	                    "EV2.2_FECHADA" = TRUE AND "EV4.2_FECHADA" = TRUE AND
	                    "EV5.2_FECHADA" = TRUE AND
	                    
	                    "EV1.2_FECHADA" = FALSE AND "EV3.2_FECHADA" = FALSE AND
	                    "EV2.2_ABERTA" = FALSE AND "EV4.2_ABERTA" = FALSE AND
	                    "EV5.2_ABERTA" = FALSE
	                THEN
	                    "Dados_Ciclo".POS_EVS_FILT_2 := 'ESVAZIAMENTO';
	                ELSE
	                    
	                    IF "EV1.2_FECHADA" = TRUE AND "EV2.2_FECHADA" = TRUE AND
	                        "EV3.2_FECHADA" = TRUE AND "EV4.2_FECHADA" = TRUE AND
	                        "EV5.2_FECHADA" = TRUE AND
	                        
	                        "EV1.2_ABERTA" = FALSE AND "EV2.2_ABERTA" = FALSE AND
	                        "EV3.2_ABERTA" = FALSE AND "EV4.2_ABERTA" = FALSE AND
	                        "EV5.2_ABERTA" = FALSE
	                    THEN
	                        "Dados_Ciclo".POS_EVS_FILT_2 := 'FECHO';
	                    ELSE
	                        "Dados_Ciclo".POS_EVS_FILT_2 := 'NULL';
	                    END_IF;
	                END_IF;
	            END_IF;
	        END_IF;
	    END_IF;
	    
	END_REGION
	
	//Envio de estado de avaria para hmi
	//conversão de clock para piscar quando ocorre avaria de EVs
	#"temp_clock_0.625Hz" := BOOL_TO_INT("Clock_0.625Hz");
	
	//FILTRO 1
	REGION Estado_EV1.1
	    "T_ABERTURA_EV1.1_HMI".TON(IN := "EV1.1",                   //Quando EV1.1 recebe sinal para abrir, inicia uma contagem
	   PT := "Inputs_HMI".T_POS_EVS);
	    
	    "T_FECHO_EV1.1_HMI".TON(IN := NOT "EV1.1",                  //Quando EV1.1 recebe sinal para fechar, inicia uma contagem
	   PT := "Inputs_HMI".T_POS_EVS);
	                                                                //No final da contagem avalia se a EV está na posição pretendida
	                                                                
	    IF ("T_ABERTURA_EV1.1_HMI".Q AND (NOT "EV1.1_ABERTA" OR ("EV1.1_ABERTA" AND "EV1.1_FECHADA"))) OR   //Condição de avaria
	        ("T_FECHO_EV1.1_HMI".Q AND (NOT "EV1.1_FECHADA" OR ("EV1.1_ABERTA" AND "EV1.1_FECHADA"))) THEN  //para evitar dois estados 
	       #"avaria_ev1.1" := TRUE;                                                                     //na pagcmd evs da hmi
	    ELSE
	       #"avaria_ev1.1" := FALSE;
	    END_IF;
	    
	    
	    IF #"avaria_ev1.1" = FALSE AND "EV1.1_ABERTA" AND NOT "EV1.1_FECHADA" THEN //Condição de EV1.1 ABERTA
	        "Estados_HMI"."EV1.1_ESTADO" := 1;
	        "Estados_HMI"."EV1.1_ESTADO_PAGCMD" := 1;
	    END_IF;
	    
	    
	    IF #"avaria_ev1.1" = FALSE AND "EV1.1_FECHADA" AND NOT "EV1.1_ABERTA" THEN //Condição de EV1.1 Fechada
	        "Estados_HMI"."EV1.1_ESTADO" := 0;
	        "Estados_HMI"."EV1.1_ESTADO_PAGCMD" := 0;
	    END_IF;
	    
	    
	    IF ("T_ABERTURA_EV1.1_HMI".Q AND (NOT "EV1.1_ABERTA" OR ("EV1.1_ABERTA" AND "EV1.1_FECHADA"))) OR   //Condição de avaria
	        ("T_FECHO_EV1.1_HMI".Q AND (NOT "EV1.1_FECHADA" OR ("EV1.1_ABERTA" AND "EV1.1_FECHADA"))) THEN
	        
	        "Estados_HMI"."EV1.1_ESTADO_PAGCMD" := 2;
	        
	        CASE #"temp_clock_0.625Hz" OF
	            0:
	                "Estados_HMI"."EV1.1_ESTADO" := 0;
	                
	            1:
	                "Estados_HMI"."EV1.1_ESTADO" := 2;
	        END_CASE;
	    END_IF;
	    
	    IF "T_ABERTURA_EV1.1_HMI".Q = FALSE AND "T_FECHO_EV1.1_HMI".Q = FALSE AND
	        "EV1.1_ABERTA" = FALSE AND "EV1.1_FECHADA" = FALSE THEN  //Condição de transição das EVs
	        
	        "Estados_HMI"."EV1.1_ESTADO_PAGCMD" := 3;
	        
	        CASE #"temp_clock_0.625Hz" OF
	            0:
	                "Estados_HMI"."EV1.1_ESTADO" := 0;
	            1:
	                "Estados_HMI"."EV1.1_ESTADO" := 3;
	        END_CASE;
	    END_IF;
	    
	END_REGION
	
	REGION Estado_EV2.1
	    
	    "T_ABERTURA_EV2.1_HMI".TON(IN := "EV2.1",                   //Quando EV2.1 recebe sinal para abrir, inicia uma contagem
	                               PT := "Inputs_HMI".T_POS_EVS);
	    
	    "T_FECHO_EV2.1_HMI".TON(IN := NOT "EV2.1",                  //Quando EV2.1 recebe sinal para fechar, inicia uma contagem
	                            PT := "Inputs_HMI".T_POS_EVS);
	                                                                //No final da contagem avalia se a EV está na posição pretendida
	                                                                
	    IF ("T_ABERTURA_EV2.1_HMI".Q AND (NOT "EV2.1_ABERTA" OR ("EV2.1_ABERTA" AND "EV2.1_FECHADA"))) OR   //Condição de avaria
	        ("T_FECHO_EV2.1_HMI".Q AND (NOT "EV2.1_FECHADA" OR ("EV2.1_ABERTA" AND "EV2.1_FECHADA"))) THEN
	        #"avaria_ev2.1" := TRUE;
	    ELSE
	        #"avaria_ev2.1" := FALSE;
	    END_IF;
	    
	                                                                
	    IF #"avaria_ev2.1" = FALSE AND"EV2.1_ABERTA" AND NOT "EV2.1_FECHADA" THEN //Condição de EV2.1 ABERTA
	        "Estados_HMI"."EV2.1_ESTADO" := 1;
	        "Estados_HMI"."EV2.1_ESTADO_PAGCMD" := 1;
	    END_IF;
	    
	    
	    IF #"avaria_ev2.1" = FALSE AND"EV2.1_FECHADA" AND NOT "EV2.1_ABERTA" THEN //Condição de EV2.1 Fechada
	        "Estados_HMI"."EV2.1_ESTADO" := 0;
	        "Estados_HMI"."EV2.1_ESTADO_PAGCMD" := 0;
	    END_IF;
	    
	    
	    IF ("T_ABERTURA_EV2.1_HMI".Q AND (NOT "EV2.1_ABERTA" OR ("EV2.1_ABERTA" AND "EV2.1_FECHADA"))) OR   //Condição de avaria
	        ("T_FECHO_EV2.1_HMI".Q AND (NOT "EV2.1_FECHADA" OR ("EV2.1_ABERTA" AND "EV2.1_FECHADA"))) THEN
	        
	        "Estados_HMI"."EV2.1_ESTADO_PAGCMD" := 2;
	        
	        CASE #"temp_clock_0.625Hz" OF
	            0:
	                "Estados_HMI"."EV2.1_ESTADO" := 0;
	            1:
	                "Estados_HMI"."EV2.1_ESTADO" := 2;
	        END_CASE;
	    END_IF;
	    
	    IF "T_ABERTURA_EV2.1_HMI".Q = FALSE AND "T_FECHO_EV2.1_HMI".Q = FALSE AND
	        "EV2.1_ABERTA" = FALSE AND "EV2.1_FECHADA" = FALSE THEN  //Condição de transição das EVs
	        
	        "Estados_HMI"."EV2.1_ESTADO_PAGCMD" := 3;
	        
	        CASE #"temp_clock_0.625Hz" OF
	            0:
	                "Estados_HMI"."EV2.1_ESTADO" := 0;
	            1:
	                "Estados_HMI"."EV2.1_ESTADO" := 3;
	        END_CASE;
	    END_IF;
	                                                                
	END_REGION
	
	REGION Estado_EV3.1
	    
	    "T_ABERTURA_EV3.1_HMI".TON(IN := "EV3.1",                   //Quando EV3.1 recebe sinal para abrir, inicia uma contagem
	                               PT := "Inputs_HMI".T_POS_EVS);
	    
	    "T_FECHO_EV3.1_HMI".TON(IN := NOT "EV3.1",                  //Quando EV3.1 recebe sinal para fechar, inicia uma contagem
	                            PT := "Inputs_HMI".T_POS_EVS);
	    //No final da contagem avalia se a EV está na posição pretendida
	    
	    IF ("T_ABERTURA_EV3.1_HMI".Q AND (NOT "EV3.1_ABERTA" OR ("EV3.1_ABERTA" AND "EV3.1_FECHADA"))) OR   //Condição de avaria
	        ("T_FECHO_EV3.1_HMI".Q AND (NOT "EV3.1_FECHADA" OR ("EV3.1_ABERTA" AND "EV3.1_FECHADA"))) THEN
	        #"avaria_ev3.1" := TRUE;
	    ELSE
	        #"avaria_ev3.1" := FALSE;
	    END_IF;
	    
	    
	    IF #"avaria_ev3.1" = FALSE AND "EV3.1_ABERTA" AND NOT "EV3.1_FECHADA" THEN //Condição de EV3.1 ABERTA
	        "Estados_HMI"."EV3.1_ESTADO" := 1;
	        "Estados_HMI"."EV3.1_ESTADO_PAGCMD" := 1;
	    END_IF;
	    
	    
	    IF #"avaria_ev3.1" = FALSE AND "EV3.1_FECHADA" AND NOT "EV3.1_ABERTA" THEN //Condição de EV3.1 Fechada
	        "Estados_HMI"."EV3.1_ESTADO" := 0;
	        "Estados_HMI"."EV3.1_ESTADO_PAGCMD" := 0;
	    END_IF;
	    
	    
	    IF ("T_ABERTURA_EV3.1_HMI".Q AND (NOT "EV3.1_ABERTA" OR ("EV3.1_ABERTA" AND "EV3.1_FECHADA"))) OR   //Condição de avaria
	        ("T_FECHO_EV3.1_HMI".Q AND (NOT "EV3.1_FECHADA" OR ("EV3.1_ABERTA" AND "EV3.1_FECHADA"))) THEN
	        
	        "Estados_HMI"."EV3.1_ESTADO_PAGCMD" := 2;
	        
	        CASE #"temp_clock_0.625Hz" OF
	            0:
	                "Estados_HMI"."EV3.1_ESTADO" := 0;
	            1:
	                "Estados_HMI"."EV3.1_ESTADO" := 2;
	        END_CASE;
	    END_IF;
	    
	    IF "T_ABERTURA_EV3.1_HMI".Q = FALSE AND "T_FECHO_EV3.1_HMI".Q = FALSE AND
	        "EV3.1_ABERTA" = FALSE AND "EV3.1_FECHADA" = FALSE THEN  //Condição de transição das EVs
	        
	        "Estados_HMI"."EV3.1_ESTADO_PAGCMD" := 3;
	        
	        CASE #"temp_clock_0.625Hz" OF
	            0:
	                "Estados_HMI"."EV3.1_ESTADO" := 0;
	            1:
	                "Estados_HMI"."EV3.1_ESTADO" := 3;
	        END_CASE;
	    END_IF;
	    
	END_REGION
	
	REGION Estado_EV4.1
	    
	    "T_ABERTURA_EV4.1_HMI".TON(IN := "EV4.1",                   //Quando EV4.1 recebe sinal para abrir, inicia uma contagem
	                               PT := "Inputs_HMI".T_POS_EVS);
	    
